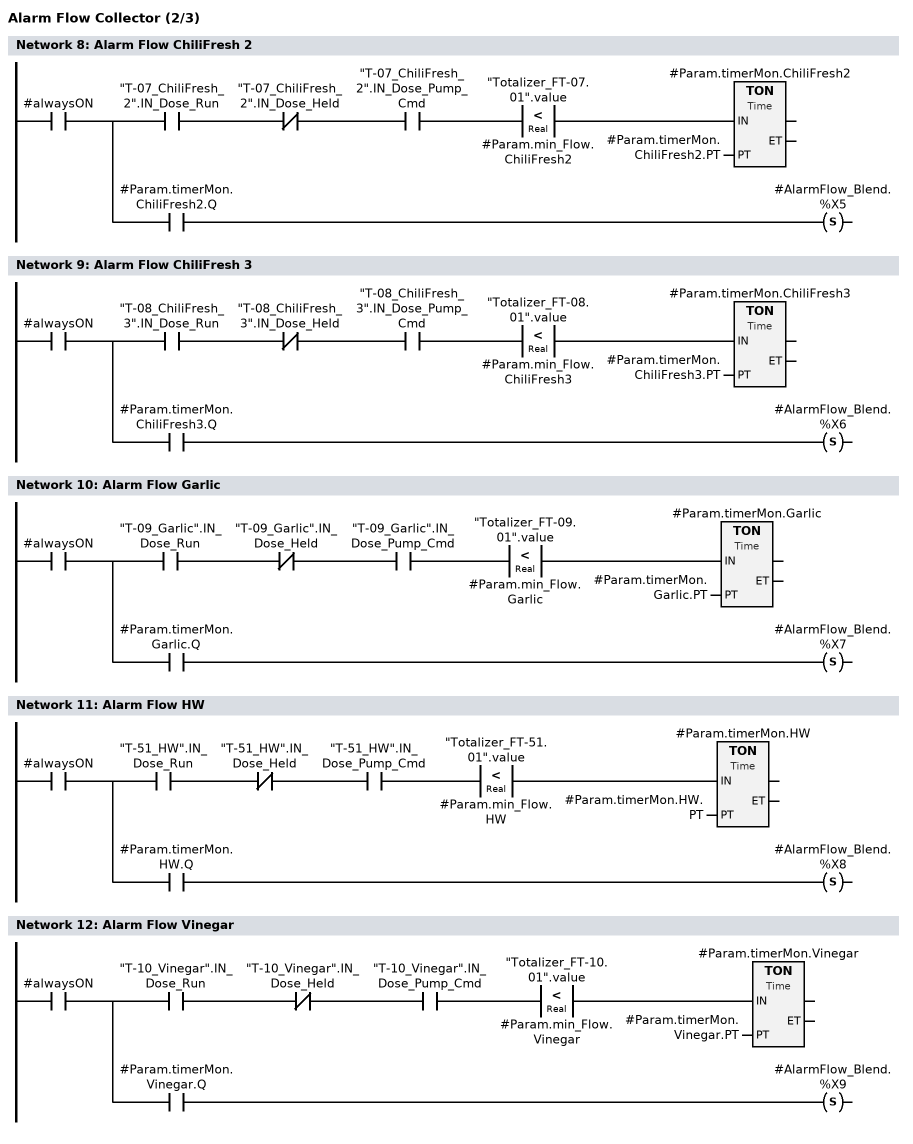
   RUNG wire#powerrail
      Contact( #alwaysON )
      wire#w1
      Contact( "T-07_ChiliFresh_2".IN_Dose_Run )
      I_Contact( "T-07_ChiliFresh_2".IN_Dose_Held )
      Contact( "T-07_ChiliFresh_2".IN_Dose_Pump_Cmd )
      { S7_Templates := "SrcType := Real" } LT_Contact(in1 := "Totalizer_FT-07.01".value, in2 := #Param.min_Flow.ChiliFresh2)
      { S7_Templates := "time_type := Time" } #Param.timerMon.ChiliFresh2.TON(pt := #Param.timerMon.ChiliFresh2.PT, et =>)
   END_RUNG
   RUNG wire#w1
      Contact( #Param.timerMon.ChiliFresh2.Q )
      S_Coil( #AlarmFlow_Blend.%X5 )
   END_RUNG
   // the same network as SCL:
   #Param.timerMon.ChiliFresh2.TON(IN := #alwaysON AND "T-07_ChiliFresh_2".IN_Dose_Run AND NOT "T-07_ChiliFresh_2".IN_Dose_Held AND "T-07_ChiliFresh_2".IN_Dose_Pump_Cmd AND ("Totalizer_FT-07.01".value < #Param.min_Flow.ChiliFresh2),
                           PT := #Param.timerMon.ChiliFresh2.PT);
   IF #alwaysON AND #Param.timerMon.ChiliFresh2.Q THEN #AlarmFlow_Blend.%X5 := TRUE; END_IF;
END_REGION

REGION Network 9: Alarm Flow ChiliFresh 3
   RUNG wire#powerrail
      Contact( #alwaysON )
      wire#w1
      Contact( "T-08_ChiliFresh_3".IN_Dose_Run )
      I_Contact( "T-08_ChiliFresh_3".IN_Dose_Held )
      Contact( "T-08_ChiliFresh_3".IN_Dose_Pump_Cmd )
      { S7_Templates := "SrcType := Real" } LT_Contact(in1 := "Totalizer_FT-08.01".value, in2 := #Param.min_Flow.ChiliFresh3)
      { S7_Templates := "time_type := Time" } #Param.timerMon.ChiliFresh3.TON(pt := #Param.timerMon.ChiliFresh3.PT, et =>)
   END_RUNG
   RUNG wire#w1
      Contact( #Param.timerMon.ChiliFresh3.Q )
      S_Coil( #AlarmFlow_Blend.%X6 )
   END_RUNG
   // the same network as SCL:
   #Param.timerMon.ChiliFresh3.TON(IN := #alwaysON AND "T-08_ChiliFresh_3".IN_Dose_Run AND NOT "T-08_ChiliFresh_3".IN_Dose_Held AND "T-08_ChiliFresh_3".IN_Dose_Pump_Cmd AND ("Totalizer_FT-08.01".value < #Param.min_Flow.ChiliFresh3),
                           PT := #Param.timerMon.ChiliFresh3.PT);
   IF #alwaysON AND #Param.timerMon.ChiliFresh3.Q THEN #AlarmFlow_Blend.%X6 := TRUE; END_IF;
END_REGION

REGION Network 10: Alarm Flow Garlic
   RUNG wire#powerrail
      Contact( #alwaysON )
      wire#w1
      Contact( "T-09_Garlic".IN_Dose_Run )
      I_Contact( "T-09_Garlic".IN_Dose_Held )
      Contact( "T-09_Garlic".IN_Dose_Pump_Cmd )
      { S7_Templates := "SrcType := Real" } LT_Contact(in1 := "Totalizer_FT-09.01".value, in2 := #Param.min_Flow.Garlic)
      { S7_Templates := "time_type := Time" } #Param.timerMon.Garlic.TON(pt := #Param.timerMon.Garlic.PT, et =>)
   END_RUNG
   RUNG wire#w1
      Contact( #Param.timerMon.Garlic.Q )
      S_Coil( #AlarmFlow_Blend.%X7 )
   END_RUNG
   // the same network as SCL:
   #Param.timerMon.Garlic.TON(IN := #alwaysON AND "T-09_Garlic".IN_Dose_Run AND NOT "T-09_Garlic".IN_Dose_Held AND "T-09_Garlic".IN_Dose_Pump_Cmd AND ("Totalizer_FT-09.01".value < #Param.min_Flow.Garlic),
                           PT := #Param.timerMon.Garlic.PT);
   IF #alwaysON AND #Param.timerMon.Garlic.Q THEN #AlarmFlow_Blend.%X7 := TRUE; END_IF;
END_REGION

REGION Network 11: Alarm Flow HW
   RUNG wire#powerrail
      Contact( #alwaysON )
      wire#w1
      Contact( "T-51_HW".IN_Dose_Run )
      I_Contact( "T-51_HW".IN_Dose_Held )
      Contact( "T-51_HW".IN_Dose_Pump_Cmd )
      { S7_Templates := "SrcType := Real" } LT_Contact(in1 := "Totalizer_FT-51.01".value, in2 := #Param.min_Flow.HW)
      { S7_Templates := "time_type := Time" } #Param.timerMon.HW.TON(pt := #Param.timerMon.HW.PT, et =>)
   END_RUNG
   RUNG wire#w1
      Contact( #Param.timerMon.HW.Q )
      S_Coil( #AlarmFlow_Blend.%X8 )
   END_RUNG
   // the same network as SCL:
   #Param.timerMon.HW.TON(IN := #alwaysON AND "T-51_HW".IN_Dose_Run AND NOT "T-51_HW".IN_Dose_Held AND "T-51_HW".IN_Dose_Pump_Cmd AND ("Totalizer_FT-51.01".value < #Param.min_Flow.HW),
                          PT := #Param.timerMon.HW.PT);
   IF #alwaysON AND #Param.timerMon.HW.Q THEN #AlarmFlow_Blend.%X8 := TRUE; END_IF;
END_REGION

REGION Network 12: Alarm Flow Vinegar
   RUNG wire#powerrail
      Contact( #alwaysON )
      wire#w1
      Contact( "T-10_Vinegar".IN_Dose_Run )
      I_Contact( "T-10_Vinegar".IN_Dose_Held )
      Contact( "T-10_Vinegar".IN_Dose_Pump_Cmd )
      { S7_Templates := "SrcType := Real" } LT_Contact(in1 := "Totalizer_FT-10.01".value, in2 := #Param.min_Flow.Vinegar)
      { S7_Templates := "time_type := Time" } #Param.timerMon.Vinegar.TON(pt := #Param.timerMon.Vinegar.PT, et =>)
   END_RUNG
   RUNG wire#w1
      Contact( #Param.timerMon.Vinegar.Q )
      S_Coil( #AlarmFlow_Blend.%X9 )
   END_RUNG
   // the same network as SCL:
   #Param.timerMon.Vinegar.TON(IN := #alwaysON AND "T-10_Vinegar".IN_Dose_Run AND NOT "T-10_Vinegar".IN_Dose_Held AND "T-10_Vinegar".IN_Dose_Pump_Cmd AND ("Totalizer_FT-10.01".value < #Param.min_Flow.Vinegar),
                           PT := #Param.timerMon.Vinegar.PT);
   IF #alwaysON AND #Param.timerMon.Vinegar.Q THEN #AlarmFlow_Blend.%X9 := TRUE; END_IF;
END_REGION

REGION Network 13: Alarm Flow Sugar
END_REGION

REGION Network 14: Alarm Flow Salt
END_REGION

REGION Network 15: Alarm Flow Prowater
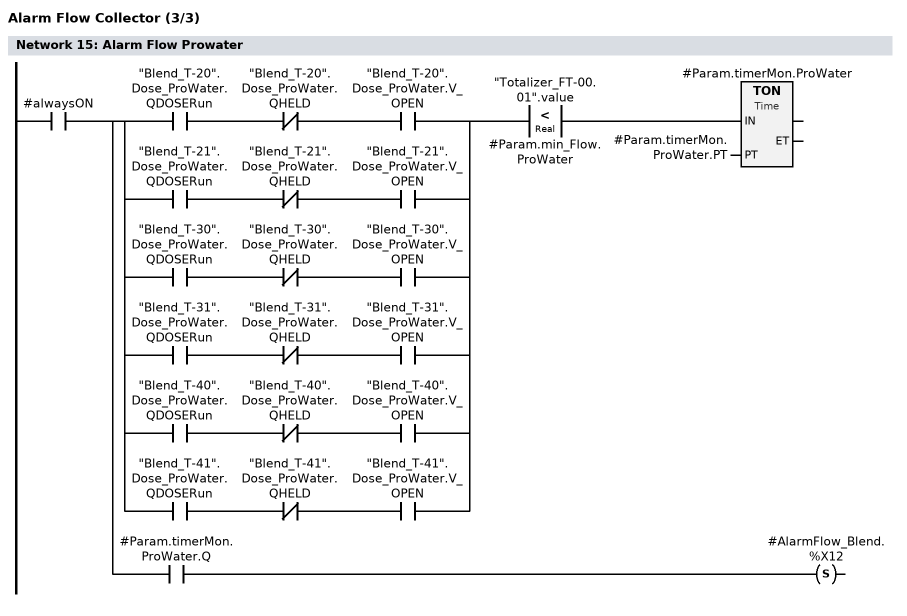
   RUNG wire#powerrail
      Contact( #alwaysON )
      wire#w1
      Contact( "Blend_T-20".Dose_ProWater.QDOSERun )
      I_Contact( "Blend_T-20".Dose_ProWater.QHELD )
      Contact( "Blend_T-20".Dose_ProWater.V_OPEN )
      wire#w2
      { S7_Templates := "SrcType := Real" } LT_Contact(in1 := "Totalizer_FT-00.01".value, in2 := #Param.min_Flow.ProWater)
      { S7_Templates := "time_type := Time" } #Param.timerMon.ProWater.TON(pt := #Param.timerMon.ProWater.PT, et =>)
   END_RUNG
   RUNG wire#w1
      Contact( "Blend_T-21".Dose_ProWater.QDOSERun )
      I_Contact( "Blend_T-21".Dose_ProWater.QHELD )
      Contact( "Blend_T-21".Dose_ProWater.V_OPEN )
   END_RUNG wire#w2
   RUNG wire#w1
      Contact( "Blend_T-30".Dose_ProWater.QDOSERun )
      I_Contact( "Blend_T-30".Dose_ProWater.QHELD )
      Contact( "Blend_T-30".Dose_ProWater.V_OPEN )
   END_RUNG wire#w2
   RUNG wire#w1
      Contact( "Blend_T-31".Dose_ProWater.QDOSERun )
      I_Contact( "Blend_T-31".Dose_ProWater.QHELD )
      Contact( "Blend_T-31".Dose_ProWater.V_OPEN )
   END_RUNG wire#w2
   RUNG wire#w1
      Contact( "Blend_T-40".Dose_ProWater.QDOSERun )
      I_Contact( "Blend_T-40".Dose_ProWater.QHELD )
      Contact( "Blend_T-40".Dose_ProWater.V_OPEN )
   END_RUNG wire#w2
   RUNG wire#w1
      Contact( "Blend_T-41".Dose_ProWater.QDOSERun )
      I_Contact( "Blend_T-41".Dose_ProWater.QHELD )
      Contact( "Blend_T-41".Dose_ProWater.V_OPEN )
   END_RUNG wire#w2
   RUNG wire#w1
      Contact( #Param.timerMon.ProWater.Q )
      S_Coil( #AlarmFlow_Blend.%X12 )
   END_RUNG
   // the same network as SCL:
   #Param.timerMon.ProWater.TON(IN := #alwaysON AND (("Blend_T-20".Dose_ProWater.QDOSERun AND NOT "Blend_T-20".Dose_ProWater.QHELD AND "Blend_T-20".Dose_ProWater.V_OPEN) OR ("Blend_T-21".Dose_ProWater.QDOSERun AND NOT "Blend_T-21".Dose_ProWater.QHELD AND "Blend_T-21".Dose_ProWater.V_OPEN) OR ("Blend_T-30".Dose_ProWater.QDOSERun AND NOT "Blend_T-30".Dose_ProWater.QHELD AND "Blend_T-30".Dose_ProWater.V_OPEN) OR ("Blend_T-31".Dose_ProWater.QDOSERun AND NOT "Blend_T-31".Dose_ProWater.QHELD AND "Blend_T-31".Dose_ProWater.V_OPEN) OR ("Blend_T-40".Dose_ProWater.QDOSERun AND NOT "Blend_T-40".Dose_ProWater.QHELD AND "Blend_T-40".Dose_ProWater.V_OPEN) OR ("Blend_T-41".Dose_ProWater.QDOSERun AND NOT "Blend_T-41".Dose_ProWater.QHELD AND "Blend_T-41".Dose_ProWater.V_OPEN)) AND ("Totalizer_FT-00.01".value < #Param.min_Flow.ProWater),
                           PT := #Param.timerMon.ProWater.PT);
   IF #alwaysON AND #Param.timerMon.ProWater.Q THEN #AlarmFlow_Blend.%X12 := TRUE; END_IF;
END_REGION
END_FUNCTION_BLOCK

FUNCTION_BLOCK "Blend_Tank"   // FB210, LAD
{ S7_Optimized_Access := 'TRUE' }
VERSION : 0.1
// stored: AutoNumber false, IsIECCheckEnabled false, IsRetainMemResEnabled false, MemoryReserve 100, SetENOAutomatically false, UDAEnableTagReadback false
   VAR_INPUT
      IN_FBAV_Header1 : Bool;
      IN_FBAV_Header2 : Bool;
      IN_FBAV_Vinegar : Bool;
      IN_FBAV_Sugar : Bool;
      IN_FBAV_Salt : Bool;
      IN_FBAV_ProWater : Bool;
      IN_FBAV_Homomixer : Bool;
      IN_FBAV_Transfer1 : Bool;
      IN_FBAV_Transfer2 : Bool;
      IN_FBAV_Transfer3 : Bool;
      IN_FBAV_Outlet : Bool;
      IN_FBAV_CIP : Bool;
      IN_FBP_Transfer1 : Bool;
      IN_FBP_Transfer1_Sp : Real;
      IN_FBP_Transfer2 : Bool;
      IN_FBP_Transfer2_Sp : Real;
      IN_FBP_Transfer3 : Bool;
      IN_FBP_Transfer3_Sp : Real;
      IN_FBP_CIP : Bool;
      IN_FBP_CIP_Sp : Real;
      IN_LT01 : Real;
      "BFT-1 Prod Req" : Bool;
      "BFT-1 Prod Line" : Bool;
      "BFT-1 CIP Enable" : Bool;
      "BFT-1 CIPLine" : Bool;
      "BFT-2 Prod Req" : Bool;
      "BFT-2 Prod Line" : Bool;
      "BFT-2 CIP Enable" : Bool;
      "BFT-2 CIPLine" : Bool;
      "BFT-3 Prod Req" : Bool;
      "BFT-3 Prod Line" : Bool;
      "BFT-3 CIP Enable" : Bool;
      "BFT-3 CIPLine" : Bool;
      "Transfer 1 Busy" : Bool;
      "Transfer 2 Busy" : Bool;
      "Transfer 3 Busy" : Bool;
      "Header 1 Available" : Bool;   // Header 1 line free
      "Header 2 Available" : Bool;   // Header 2 line free
      "Vinegar Available" : Bool;   // Vinegar line free
      "Sugar Available" : Bool;   // Sugar line free
      "Salt Available" : Bool;   // Salt line free
      "ProWater Available" : Bool;   // ProWater line free
      "Homomixer Available" : Bool;   // Homomixer line free
      IN_LDT : Date_And_Time;
      "CIP Pulse" : Bool;
      "CIP Supply ON" : Bool;
      "CIP Req OK" : Bool;
      "CIP Complete" : Bool;
      "CIP Busy" : Bool;
   END_VAR
   VAR_OUTPUT
      Out_AV_Header1 : Bool;
      Out_AV_Header2 : Bool;
      Out_AV_Vinegar : Bool;
      Out_AV_Sugar : Bool;
      Out_AV_Salt : Bool;
      Out_AV_ProWater : Bool;
      Out_AV_Homomixer : Bool;
      Out_AV_Transfer1 : Bool;
      Out_AV_Transfer2 : Bool;
      Out_AV_Transfer3 : Bool;
      Out_AV_Outlet : Bool;
      Out_AV_CIP : Bool;
      Out_P_Transfer1 : Bool;
      Out_P_Transfer1_Sp : Real;
      Out_P_Transfer2 : Bool;
      Out_P_Transfer2_Sp : Real;
      Out_P_Transfer3 : Bool;
      Out_P_Transfer3_Sp : Real;
      Out_P_CIP : Bool;
      Out_P_CIP_Sp : Real;
      Out_Agi : Bool;
      Out_Agi_Sp : Real;
      "Header 1 Req" : Bool;
      "Header 2 Req" : Bool;
      "Vinegar Req" : Bool;
      "Sugar Req" : Bool;
      "Salt Req" : Bool;
      "ProWater Req" : Bool;
      "Homomixer Req" : Bool;
      Out_CIP_Req : Bool;
      Out_CIP_Line_Open : Bool;
   END_VAR
   VAR
      Cmd : Struct
         "Ready For Transfer" : Bool;
         "CIP Tank 1" : Bool;
         "CIP Tank 2" : Bool;
         "CIP Line" : Bool;
         "Dose Head 1" : Bool;
         "Dose Head 2" : Bool;
         Agitator_Mode : Bool;   // 0: Speed Fix, 1: Speed by level
      END_STRUCT;
   END_VAR
   VAR RETAIN
      Param : Struct
         SP_Level_LL : Real := 10.0;
         SP_Level_ML : Real := 80.0;
         SP_Level_HL : Real := 100.0;
         L_Hi_Lim : Real := 100.0;
         L_Lo_Lim : Real := 0.0;
         L_Hys : Real := 2.0;
         LB_ON : Real := 20.0;
         LB_OFF : Real := 17.0;
         LB1_ON : Real := 15.0;
         LB1_OFF : Real := 10.0;
         LB2_ON : Real := 35.0;
         LB2_OFF : Real := 30.0;
         LB3_ON : Real := 65.0;
         LB3_OFF : Real := 60.0;
         SP_P1_Speed : Real := 80.0;
         SP_P2_Speed : Real := 80.0;
         SP_P3_Speed : Real := 80.0;
         SP_LB_Speed : Real := 50.0;
         SP_LB1_Speed : Real := 25.0;
         SP_LB2_Speed : Real := 50.0;
         SP_LB3_Speed : Real := 80.0;
         CIP_Tank_P_Ret_Speed : Real := 60.0;
         CIP_Ret_ON_SP : Real := 10.0;
         CIP_Ret_OFF_SP : Real := 0.0;
         Flushing_HW_Timer : Time := T#60s;
      END_STRUCT;
   END_VAR
   VAR
      State : Struct
         "Tank LL" : Bool;
         "Tank ML" : Bool;
         "Tank HL" : Bool;
         LB_ON : Bool;
         LB1_ON : Bool;
         LB2_ON : Bool;
         LB3_ON : Bool;
         "CIP Tank" : Bool;
         "CIP Tank Ena" : Bool;
         "CIP Tank Ret 1 Ena" : Bool;
         "CIP Tank Ret 2 Ena" : Bool;
         "CIP Line" : Bool;
         "CIP Line Ena" : Bool;
         "CIP Return On" : Bool;
         "Dose On Prog" : Bool;
         "Dose EN" : Bool;
         "Ready For Transfer" : Bool;
         "Ready For Transfer Ena" : Bool;
         "BFT-1 EN" : Bool;
         "BFT-2 EN" : Bool;
         "BFT-3 EN" : Bool;
         "RM Dose" : Bool;
         "Transfer 1 On Progress" : Bool;
         "Transfer 2 On Progress" : Bool;
         "Transfer 3 On Progress" : Bool;
         "DoseHead1 ON" : Bool;
         "DoseHead2 ON" : Bool;
      END_STRUCT;
      Dose : Struct
         Dose_Start : DWord;
         Dose_Pause : DWord;
         Dose_Stop : DWord;
         Dose_State : DWord;
         Dose_Tank_Available : Word;
         Dose_Prod_Ready : Word;
         Dose_Header_Req : DWord;
         Dose_EN : Word;
      END_STRUCT;
      "Dose_Level_%" : Struct
         "ChiliAwetan1%" : Real;
         "ChiliAwetan2%" : Real;
         "ChiliAwetan3%" : Real;
         "Tomato%" : Real;
         "ChiliFresh1%" : Real;
         "ChiliFresh2%" : Real;
         "ChiliFresh3%" : Real;
         "Garlic%" : Real;
         "HW%" : Real;
         "Vinegar%" : Real;
         "Sugar%" : Real;
         "Salt%" : Real;
         "ProWater%" : Real;
         "Homomixer%" : Real;
      END_STRUCT;
      Dose_Level_Lit : Struct
         ChiliAwetan1Lit : Real;
         ChiliAwetan2Lit : Real;
         ChiliAwetan3Lit : Real;
         TomatoLit : Real;
         ChiliFresh1Lit : Real;
         ChiliFresh2Lit : Real;
         ChiliFresh3Lit : Real;
         GarlicLit : Real;
         HWLit : Real;
         VinegarLit : Real;
         SugarLit : Real;
         SaltLit : Real;
         ProWaterLit : Real;
         HomomixerLit : Real;
      END_STRUCT;
      SP_Dose_Level : Struct
         ChiliAwetan1Lit : Real;
         ChiliAwetan2Lit : Real;
         ChiliAwetan3Lit : Real;
         TomatoLit : Real;
         ChiliFresh1Lit : Real;
         ChiliFresh2Lit : Real;
         ChiliFresh3Lit : Real;
         GarlicLit : Real;
         HWLit : Real;
         VinegarLit : Real;
         SugarLit : Real;
         SaltLit : Real;
         ProWaterLit : Real;
         HomomixerLit : Real;
      END_STRUCT;
      r : Struct
         PosE1 : Bool;
         PosE2 : Bool;
         PosE3 : Bool;
         PosE4 : Bool;
         PosE5 : Bool;
         PosE6 : Bool;
         PosE7 : Bool;
         PosE8 : Bool;
         PosE9 : Bool;
         PosE10 : Bool;
         PosE11 : Bool;
         PosE12 : Bool;
         PosE13 : Bool;
         PosE14 : Bool;
         PosE15 : Bool;
         PosE16 : Bool;
         PosE17 : Bool;
         PosE18 : Bool;
         PosE19 : Bool;
         PosE20 : Bool;
         PosE21 : Bool;
         PosE22 : Bool;
         PosE23 : Bool;
         PosE24 : Bool;
         PosE25 : Bool;
         PosE26 : Bool;
         PosE27 : Bool;
         PosE28 : Bool;
         PosE29 : Bool;
         PosE30 : Bool;
         PosE31 : Bool;
         PosE32 : Bool;
      END_STRUCT;
      Actuator : Struct
         P_Transfer1 : Bool;
         P_Transfer2 : Bool;
         P_Transfer3 : Bool;
         AV_Transfer1 : Bool;
         AV_Transfer2 : Bool;
         AV_Transfer3 : Bool;
         AV_Outlet : Bool;
         AV_CIP_Tank : Bool;
      END_STRUCT;
      SP_ChiliAwetan1 : "RawDose";
      SP_ChiliAwetan2 : "RawDose";
      SP_ChiliAwetan3 : "RawDose";
      SP_Tomato : "RawDose";
      SP_ChiliFresh1 : "RawDose";
      SP_ChiliFresh2 : "RawDose";
      SP_ChiliFresh3 : "RawDose";
      SP_Garlic : "RawDose";
      SP_HW : "Raw_Pulse";
      SP_Vinegar : "RawDose";
      SP_Sugar : "RawDose";
      SP_Salt : "RawDose";
      SP_ProWater : "Raw_Pulse";
      SP_Homomixer : "RawDose";
      Dose_ChiliAwetan1 { S7_SetPoint := 'True'} : "DOSE";
      Dose_ChiliAwetan2 { S7_SetPoint := 'True'} : "DOSE";
      Dose_ChiliAwetan3 { S7_SetPoint := 'True'} : "DOSE";
      Dose_Tomato { S7_SetPoint := 'True'} : "DOSE";
      Dose_ChiliFresh1 { S7_SetPoint := 'True'} : "DOSE";
      Dose_ChiliFresh2 { S7_SetPoint := 'True'} : "DOSE";
      Dose_ChiliFresh3 { S7_SetPoint := 'True'} : "DOSE";
      Dose_Garlic { S7_SetPoint := 'True'} : "DOSE";
      Dose_HW { S7_SetPoint := 'True'} : "DOSE";
      Dose_Vinegar { S7_SetPoint := 'True'} : "DOSE";
      Dose_Sugar { S7_SetPoint := 'True'} : "DOSE";
      Dose_Salt { S7_SetPoint := 'True'} : "DOSE";
      Dose_ProWater { S7_SetPoint := 'True'} : "DOSE";
      Dose_Homomixer { S7_SetPoint := 'True'} : "DOSE";
      AlwaysON { S7_SetPoint := 'True'} : Bool;
      L_Hys_Abs { S7_SetPoint := 'True'} : Real;
      Hys_Level_HL : Real;
      Hys_Level_ML : Real;
      Hys_Level_LL : Real;
      TimerOff_Valve_Out : TON_TIME;
      TimerOff_Valve_P_1 { S7_SetPoint := 'True'} : TON_TIME;
      TimerOff_Valve_P_2 { S7_SetPoint := 'True'} : TON_TIME;
      TimerOff_Valve_P_3 { S7_SetPoint := 'True'} : TON_TIME;
      TimerOff_Valve_P_CIP { S7_SetPoint := 'True'} : TON_TIME;
   END_VAR
   VAR RETAIN
      Last_Dose_Qty : Struct
         ChiliAwetan1 : Real;
         ChiliAwetan2 : Real;
         ChiliAwetan3 : Real;
         Tomato : Real;
         ChiliFresh1 : Real;
         ChiliFresh2 : Real;
         ChiliFresh3 : Real;
         Garlic : Real;
         HW : Real;
         Vinegar : Real;
         Sugar : Real;
         Salt : Real;
         ProWater : Real;
         Homomixer : Real;
      END_STRUCT;
   END_VAR
   VAR
      "HW Flushing" : Struct
         Status : Struct
            "Flush to Blend" : Bool;
            "Flush to Drain" : Bool;
            Drain : Bool;
            Done : Bool;
         END_STRUCT;
         Qty : Struct
            "Flush to Blend Qty" : Real;
            "Flush to Drain Qty" : Real;
            "Flush to Blend Act" : Real;
            "Flush to Drain Act" : Real;
         END_STRUCT;
         TimeDrain_SP : DInt;
         Cmd_Start_Drain : Bool;
         Cmd_Stop_Drain : Bool;
         DrainTime : TONR_TIME;
      END_STRUCT;
      PumpTF1_OnDelay : TON_TIME;
      PumpTF2_OnDelay { S7_SetPoint := 'True'} : TON_TIME;
      PumpTF3_OnDelay { S7_SetPoint := 'True'} : TON_TIME;
   END_VAR
   VAR RETAIN
      TimerON : Struct
         TimerON_1 : TON_TIME;
         TimerON_2 { S7_SetPoint := 'True'} : TON_TIME;
         TimerON_3 { S7_SetPoint := 'True'} : TON_TIME;
         TimerON_4 { S7_SetPoint := 'True'} : TON_TIME;
         TimerON_5 { S7_SetPoint := 'True'} : TON_TIME;
         TimerON_6 { S7_SetPoint := 'True'} : TON_TIME;
         TimerON_7 { S7_SetPoint := 'True'} : TON_TIME;
         TimerON_8 { S7_SetPoint := 'True'} : TON_TIME;
      END_STRUCT;
      TimerOFF : Struct
         TimerOFF_1 : TOF_TIME;
         TimerOFF_2 { S7_SetPoint := 'True'} : TOF_TIME;
         TimerOFF_3 { S7_SetPoint := 'True'} : TOF_TIME;
         TimerOFF_4 { S7_SetPoint := 'True'} : TOF_TIME;
         TimerOFF_5 { S7_SetPoint := 'True'} : TOF_TIME;
         TimerOFF_6 { S7_SetPoint := 'True'} : TOF_TIME;
         TimerOFF_7 { S7_SetPoint := 'True'} : TOF_TIME;
         TimerOFF_8 { S7_SetPoint := 'True'} : TOF_TIME;
      END_STRUCT;
   END_VAR
   // SP_ProWater.Para."SP_Qty_Fine%" := 10.0;
   // SP_Homomixer.Dose_SP := 10.0;
   // TimerON.TimerON_1.PT := T#8s;
   // TimerON.TimerON_2.PT := T#8s;
   // TimerON.TimerON_3.PT := T#10s;
   // TimerON.TimerON_4.PT := T#10s;
   // TimerON.TimerON_5.PT := T#10s;
   // TimerON.TimerON_6.PT := T#10s;
   // TimerON.TimerON_7.PT := T#10s;
   // TimerON.TimerON_8.PT := T#10s;
   // TimerOFF.TimerOFF_1.PT := T#10s;
   // TimerOFF.TimerOFF_2.PT := T#10s;
   // TimerOFF.TimerOFF_3.PT := T#10s;
   // TimerOFF.TimerOFF_4.PT := T#10s;
   // TimerOFF.TimerOFF_5.PT := T#10s;
   // TimerOFF.TimerOFF_6.PT := T#10s;
   // TimerOFF.TimerOFF_7.PT := T#10s;
   // TimerOFF.TimerOFF_8.PT := T#10s;
   VAR_TEMP   // added for the SCL form of the ladder/FBD networks
      _w1 : Bool;
      _w2 : Bool;
      _w3 : Bool;
      _w4 : Bool;
      _w5 : Bool;
      _w6 : Bool;
   END_VAR
BEGIN

REGION Network 2: Always ON
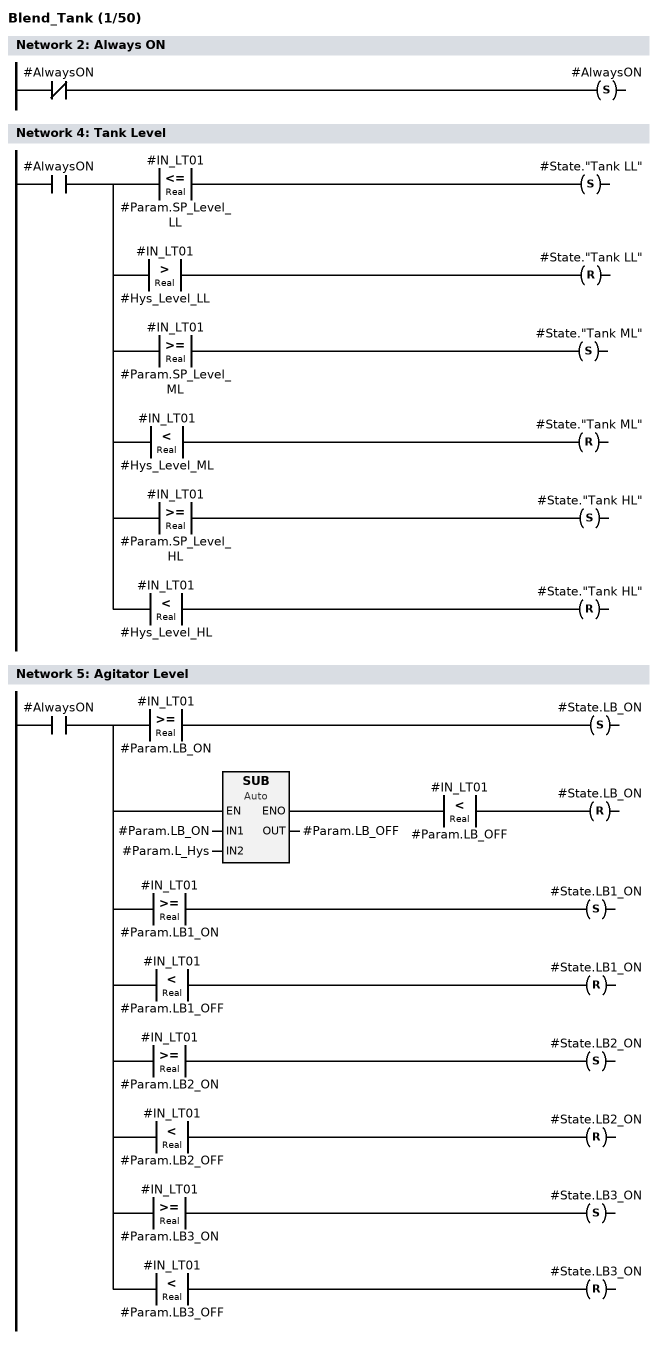
   RUNG wire#powerrail
      I_Contact( #AlwaysON )
      S_Coil( #AlwaysON )
   END_RUNG
   // the same network as SCL:
   IF NOT #AlwaysON THEN #AlwaysON := TRUE; END_IF;
END_REGION

NETWORK
TITLE = Hys Calculation
//Level Hys Absolute
      L     #Param.L_Hi_Lim;
      L     #Param.L_Lo_Lim;
      -R;
      L     100.0;
      /R;
      L     #Param.L_Hys;
      *R;
      T     #L_Hys_Abs;
//Tank High Level
      L     #Param.SP_Level_HL;
      L     #L_Hys_Abs;
      -R;
      T     #Hys_Level_HL;
//Tank Mid Level
      L     #Param.SP_Level_ML;
      L     #L_Hys_Abs;
      -R;
      T     #Hys_Level_ML;
//Tank Low Level
      L     #Param.SP_Level_LL;
      L     #L_Hys_Abs;
      +R;
      T     #Hys_Level_LL;


REGION Network 4: Tank Level
   RUNG wire#powerrail
      Contact( #AlwaysON )
      wire#w1
      { S7_Templates := "SrcType := Real" } LE_Contact(in1 := #IN_LT01, in2 := #Param.SP_Level_LL)
      S_Coil( #State."Tank LL" )
   END_RUNG
   RUNG wire#w1
      { S7_Templates := "SrcType := Real" } GT_Contact(in1 := #IN_LT01, in2 := #Hys_Level_LL)
      R_Coil( #State."Tank LL" )
   END_RUNG
   RUNG wire#w1
      { S7_Templates := "SrcType := Real" } GE_Contact(in1 := #IN_LT01, in2 := #Param.SP_Level_ML)
      S_Coil( #State."Tank ML" )
   END_RUNG
   RUNG wire#w1
      { S7_Templates := "SrcType := Real" } LT_Contact(in1 := #IN_LT01, in2 := #Hys_Level_ML)
      R_Coil( #State."Tank ML" )
   END_RUNG
   RUNG wire#w1
      { S7_Templates := "SrcType := Real" } GE_Contact(in1 := #IN_LT01, in2 := #Param.SP_Level_HL)
      S_Coil( #State."Tank HL" )
   END_RUNG
   RUNG wire#w1
      { S7_Templates := "SrcType := Real" } LT_Contact(in1 := #IN_LT01, in2 := #Hys_Level_HL)
      R_Coil( #State."Tank HL" )
   END_RUNG
   // the same network as SCL:
   IF #AlwaysON AND (#IN_LT01 <= #Param.SP_Level_LL) THEN #State."Tank LL" := TRUE; END_IF;
   IF #AlwaysON AND (#IN_LT01 > #Hys_Level_LL) THEN #State."Tank LL" := FALSE; END_IF;
   IF #AlwaysON AND (#IN_LT01 >= #Param.SP_Level_ML) THEN #State."Tank ML" := TRUE; END_IF;
   IF #AlwaysON AND (#IN_LT01 < #Hys_Level_ML) THEN #State."Tank ML" := FALSE; END_IF;
   IF #AlwaysON AND (#IN_LT01 >= #Param.SP_Level_HL) THEN #State."Tank HL" := TRUE; END_IF;
   IF #AlwaysON AND (#IN_LT01 < #Hys_Level_HL) THEN #State."Tank HL" := FALSE; END_IF;
END_REGION

REGION Network 5: Agitator Level
   RUNG wire#powerrail
      Contact( #AlwaysON )
      wire#w1
      { S7_Templates := "SrcType := Real" } GE_Contact(in1 := #IN_LT01, in2 := #Param.LB_ON)
      S_Coil( #State.LB_ON )
   END_RUNG
   RUNG wire#w1
      Sub(in1 := #Param.LB_ON, in2 := #Param.L_Hys, out => #Param.LB_OFF)
      { S7_Templates := "SrcType := Real" } LT_Contact(in1 := #IN_LT01, in2 := #Param.LB_OFF)
      R_Coil( #State.LB_ON )
   END_RUNG
   RUNG wire#w1
      { S7_Templates := "SrcType := Real" } GE_Contact(in1 := #IN_LT01, in2 := #Param.LB1_ON)
      S_Coil( #State.LB1_ON )
   END_RUNG
   RUNG wire#w1
      { S7_Templates := "SrcType := Real" } LT_Contact(in1 := #IN_LT01, in2 := #Param.LB1_OFF)
      R_Coil( #State.LB1_ON )
   END_RUNG
   RUNG wire#w1
      { S7_Templates := "SrcType := Real" } GE_Contact(in1 := #IN_LT01, in2 := #Param.LB2_ON)
      S_Coil( #State.LB2_ON )
   END_RUNG
   RUNG wire#w1
      { S7_Templates := "SrcType := Real" } LT_Contact(in1 := #IN_LT01, in2 := #Param.LB2_OFF)
      R_Coil( #State.LB2_ON )
   END_RUNG
   RUNG wire#w1
      { S7_Templates := "SrcType := Real" } GE_Contact(in1 := #IN_LT01, in2 := #Param.LB3_ON)
      S_Coil( #State.LB3_ON )
   END_RUNG
   RUNG wire#w1
      { S7_Templates := "SrcType := Real" } LT_Contact(in1 := #IN_LT01, in2 := #Param.LB3_OFF)
      R_Coil( #State.LB3_ON )
   END_RUNG
   // the same network as SCL:
   IF #AlwaysON AND (#IN_LT01 >= #Param.LB_ON) THEN #State.LB_ON := TRUE; END_IF;
   IF #AlwaysON THEN #Param.LB_OFF := #Param.LB_ON - #Param.L_Hys; END_IF;
   IF #AlwaysON AND (#IN_LT01 < #Param.LB_OFF) THEN #State.LB_ON := FALSE; END_IF;
   IF #AlwaysON AND (#IN_LT01 >= #Param.LB1_ON) THEN #State.LB1_ON := TRUE; END_IF;
   IF #AlwaysON AND (#IN_LT01 < #Param.LB1_OFF) THEN #State.LB1_ON := FALSE; END_IF;
   IF #AlwaysON AND (#IN_LT01 >= #Param.LB2_ON) THEN #State.LB2_ON := TRUE; END_IF;
   IF #AlwaysON AND (#IN_LT01 < #Param.LB2_OFF) THEN #State.LB2_ON := FALSE; END_IF;
   IF #AlwaysON AND (#IN_LT01 >= #Param.LB3_ON) THEN #State.LB3_ON := TRUE; END_IF;
   IF #AlwaysON AND (#IN_LT01 < #Param.LB3_OFF) THEN #State.LB3_ON := FALSE; END_IF;
END_REGION

REGION Network 6: Agitator ON-OFF
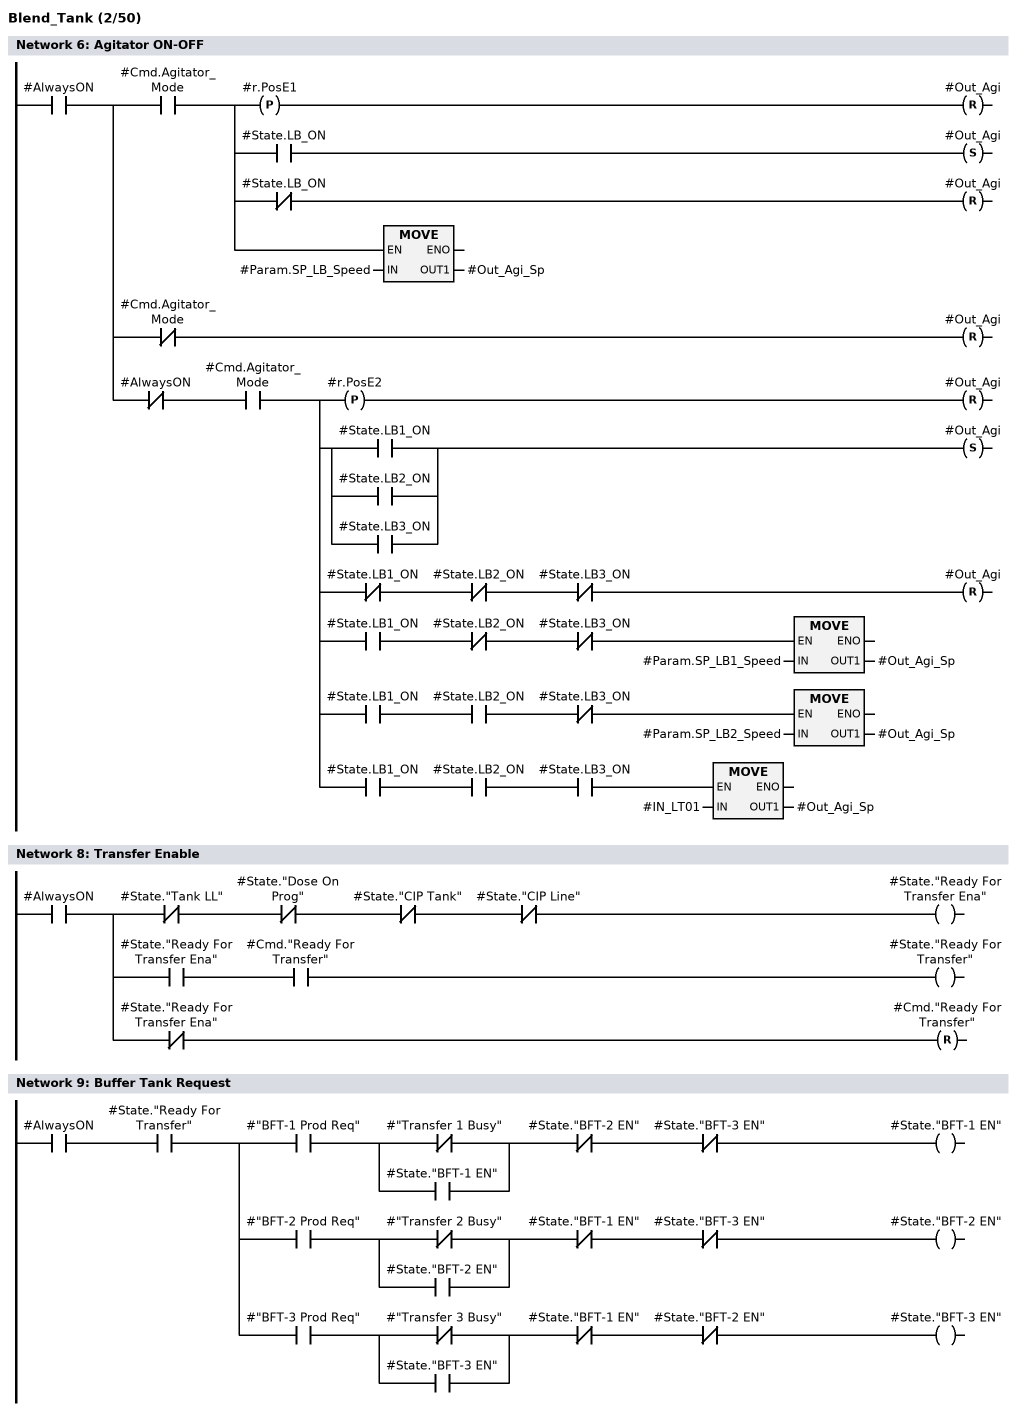
   RUNG wire#powerrail
      Contact( #AlwaysON )
      wire#w1
      Contact( #Cmd.Agitator_Mode )
      wire#w2
      P_Trig( #r.PosE1 )
      R_Coil( #Out_Agi )
   END_RUNG
   RUNG wire#w2
      Contact( #State.LB_ON )
      S_Coil( #Out_Agi )
   END_RUNG
   RUNG wire#w2
      I_Contact( #State.LB_ON )
      R_Coil( #Out_Agi )
   END_RUNG
   RUNG wire#w2
      Move(in := #Param.SP_LB_Speed, out1 => #Out_Agi_Sp)
   END_RUNG
   RUNG wire#w1
      I_Contact( #Cmd.Agitator_Mode )
      R_Coil( #Out_Agi )
   END_RUNG
   RUNG wire#w1
      I_Contact( #AlwaysON )
      Contact( #Cmd.Agitator_Mode )
      wire#w3
      P_Trig( #r.PosE2 )
      R_Coil( #Out_Agi )
   END_RUNG
   RUNG wire#w3
      Contact( #State.LB1_ON )
      wire#w4
      S_Coil( #Out_Agi )
   END_RUNG
   RUNG wire#w3
      Contact( #State.LB2_ON )
   END_RUNG wire#w4
   RUNG wire#w3
      Contact( #State.LB3_ON )
   END_RUNG wire#w4
   RUNG wire#w3
      I_Contact( #State.LB1_ON )
      I_Contact( #State.LB2_ON )
      I_Contact( #State.LB3_ON )
      R_Coil( #Out_Agi )
   END_RUNG
   RUNG wire#w3
      Contact( #State.LB1_ON )
      I_Contact( #State.LB2_ON )
      I_Contact( #State.LB3_ON )
      Move(in := #Param.SP_LB1_Speed, out1 => #Out_Agi_Sp)
   END_RUNG
   RUNG wire#w3
      Contact( #State.LB1_ON )
      Contact( #State.LB2_ON )
      I_Contact( #State.LB3_ON )
      Move(in := #Param.SP_LB2_Speed, out1 => #Out_Agi_Sp)
   END_RUNG
   RUNG wire#w3
      Contact( #State.LB1_ON )
      Contact( #State.LB2_ON )
      Contact( #State.LB3_ON )
      Move(in := #IN_LT01, out1 => #Out_Agi_Sp)
   END_RUNG
   // the same network as SCL:
   #_w1 := #AlwaysON AND #Cmd.Agitator_Mode;
   #_w2 := #_w1 AND NOT #r.PosE1;   // rising edge
   #r.PosE1 := #_w1;
   IF #_w2 THEN #Out_Agi := FALSE; END_IF;
   IF #_w1 AND #State.LB_ON THEN #Out_Agi := TRUE; END_IF;
   IF #_w1 AND NOT #State.LB_ON THEN #Out_Agi := FALSE; END_IF;
   IF #_w1 THEN #Out_Agi_Sp := #Param.SP_LB_Speed; END_IF;
   IF #AlwaysON AND NOT #Cmd.Agitator_Mode THEN #Out_Agi := FALSE; END_IF;
   #_w3 := #AlwaysON AND NOT #AlwaysON AND #Cmd.Agitator_Mode;
   #_w4 := #_w3 AND NOT #r.PosE2;   // rising edge
   #r.PosE2 := #_w3;
   IF #_w4 THEN #Out_Agi := FALSE; END_IF;
   IF #_w3 AND (#State.LB1_ON OR #State.LB2_ON OR #State.LB3_ON) THEN #Out_Agi := TRUE; END_IF;
   IF #_w3 AND NOT #State.LB1_ON AND NOT #State.LB2_ON AND NOT #State.LB3_ON THEN #Out_Agi := FALSE; END_IF;
   IF #_w3 AND #State.LB1_ON AND NOT #State.LB2_ON AND NOT #State.LB3_ON THEN
       #Out_Agi_Sp := #Param.SP_LB1_Speed;
   END_IF;
   IF #_w3 AND #State.LB1_ON AND #State.LB2_ON AND NOT #State.LB3_ON THEN
       #Out_Agi_Sp := #Param.SP_LB2_Speed;
   END_IF;
   IF #_w3 AND #State.LB1_ON AND #State.LB2_ON AND #State.LB3_ON THEN #Out_Agi_Sp := #IN_LT01; END_IF;
END_REGION

REGION Network 8: Transfer Enable
   RUNG wire#powerrail
      Contact( #AlwaysON )
      wire#w1
      I_Contact( #State."Tank LL" )
      I_Contact( #State."Dose On Prog" )
      I_Contact( #State."CIP Tank" )
      I_Contact( #State."CIP Line" )
      Coil( #State."Ready For Transfer Ena" )
   END_RUNG
   RUNG wire#w1
      Contact( #State."Ready For Transfer Ena" )
      Contact( #Cmd."Ready For Transfer" )
      Coil( #State."Ready For Transfer" )
   END_RUNG
   RUNG wire#w1
      I_Contact( #State."Ready For Transfer Ena" )
      R_Coil( #Cmd."Ready For Transfer" )
   END_RUNG
   // the same network as SCL:
   #State."Ready For Transfer Ena" := #AlwaysON AND NOT #State."Tank LL" AND NOT #State."Dose On Prog" AND NOT #State."CIP Tank" AND NOT #State."CIP Line";
   #State."Ready For Transfer" := #AlwaysON AND #State."Ready For Transfer Ena" AND #Cmd."Ready For Transfer";
   IF #AlwaysON AND NOT #State."Ready For Transfer Ena" THEN #Cmd."Ready For Transfer" := FALSE; END_IF;
END_REGION

REGION Network 9: Buffer Tank Request
   RUNG wire#powerrail
      Contact( #AlwaysON )
      Contact( #State."Ready For Transfer" )
      wire#w1
      Contact( #"BFT-1 Prod Req" )
      wire#w2
      I_Contact( #"Transfer 1 Busy" )
      wire#w3
      I_Contact( #State."BFT-2 EN" )
      I_Contact( #State."BFT-3 EN" )
      Coil( #State."BFT-1 EN" )
   END_RUNG
   RUNG wire#w2
      Contact( #State."BFT-1 EN" )
   END_RUNG wire#w3
   RUNG wire#w1
      Contact( #"BFT-2 Prod Req" )
      wire#w4
      I_Contact( #"Transfer 2 Busy" )
      wire#w5
      I_Contact( #State."BFT-1 EN" )
      I_Contact( #State."BFT-3 EN" )
      Coil( #State."BFT-2 EN" )
   END_RUNG
   RUNG wire#w4
      Contact( #State."BFT-2 EN" )
   END_RUNG wire#w5
   RUNG wire#w1
      Contact( #"BFT-3 Prod Req" )
      wire#w6
      I_Contact( #"Transfer 3 Busy" )
      wire#w7
      I_Contact( #State."BFT-1 EN" )
      I_Contact( #State."BFT-2 EN" )
      Coil( #State."BFT-3 EN" )
   END_RUNG
   RUNG wire#w6
      Contact( #State."BFT-3 EN" )
   END_RUNG wire#w7
   // the same network as SCL:
   #_w1 := #AlwaysON AND #State."Ready For Transfer";
   #State."BFT-1 EN" := #_w1 AND #"BFT-1 Prod Req" AND (NOT #"Transfer 1 Busy" OR #State."BFT-1 EN") AND NOT #State."BFT-2 EN" AND NOT #State."BFT-3 EN";
   #State."BFT-2 EN" := #_w1 AND #"BFT-2 Prod Req" AND (NOT #"Transfer 2 Busy" OR #State."BFT-2 EN") AND NOT #State."BFT-1 EN" AND NOT #State."BFT-3 EN";
   #State."BFT-3 EN" := #_w1 AND #"BFT-3 Prod Req" AND (NOT #"Transfer 3 Busy" OR #State."BFT-3 EN") AND NOT #State."BFT-1 EN" AND NOT #State."BFT-2 EN";
END_REGION

REGION Network 10: Buffer Tank Transfer Progress
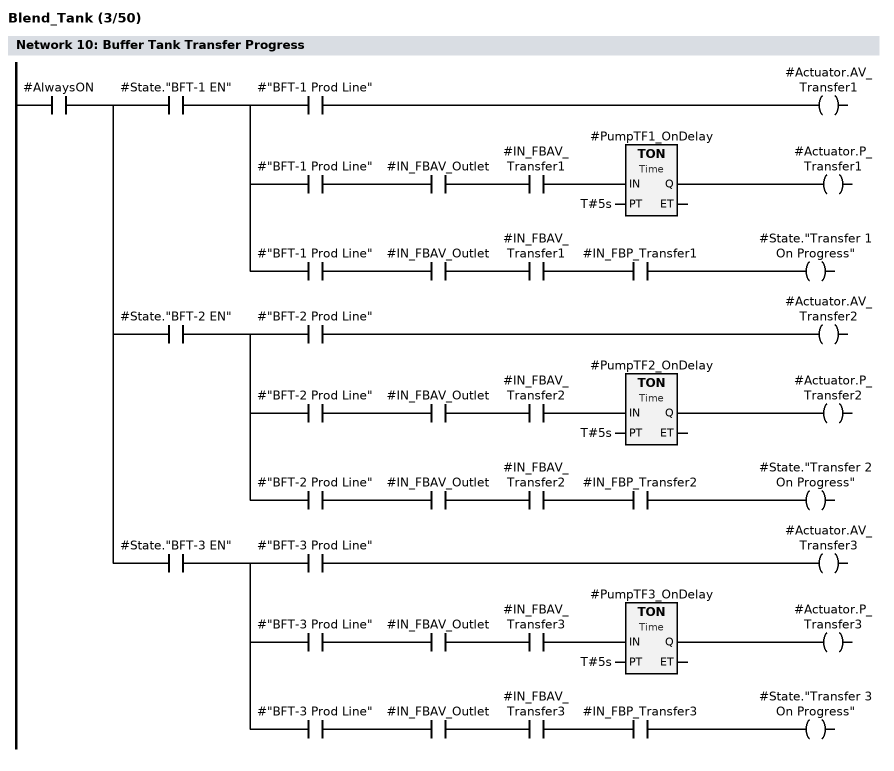
   RUNG wire#powerrail
      Contact( #AlwaysON )
      wire#w1
      Contact( #State."BFT-1 EN" )
      wire#w2
      Contact( #"BFT-1 Prod Line" )
      Coil( #Actuator.AV_Transfer1 )
   END_RUNG
   RUNG wire#w2
      Contact( #"BFT-1 Prod Line" )
      Contact( #IN_FBAV_Outlet )
      Contact( #IN_FBAV_Transfer1 )
      { S7_Templates := "time_type := Time" } #PumpTF1_OnDelay.TON(pt := T#5s, et =>)
      Coil( #Actuator.P_Transfer1 )
   END_RUNG
   RUNG wire#w2
      Contact( #"BFT-1 Prod Line" )
      Contact( #IN_FBAV_Outlet )
      Contact( #IN_FBAV_Transfer1 )
      Contact( #IN_FBP_Transfer1 )
      Coil( #State."Transfer 1 On Progress" )
   END_RUNG
   RUNG wire#w1
      Contact( #State."BFT-2 EN" )
      wire#w3
      Contact( #"BFT-2 Prod Line" )
      Coil( #Actuator.AV_Transfer2 )
   END_RUNG
   RUNG wire#w3
      Contact( #"BFT-2 Prod Line" )
      Contact( #IN_FBAV_Outlet )
      Contact( #IN_FBAV_Transfer2 )
      { S7_Templates := "time_type := Time" } #PumpTF2_OnDelay.TON(pt := T#5s, et =>)
      Coil( #Actuator.P_Transfer2 )
   END_RUNG
   RUNG wire#w3
      Contact( #"BFT-2 Prod Line" )
      Contact( #IN_FBAV_Outlet )
      Contact( #IN_FBAV_Transfer2 )
      Contact( #IN_FBP_Transfer2 )
      Coil( #State."Transfer 2 On Progress" )
   END_RUNG
   RUNG wire#w1
      Contact( #State."BFT-3 EN" )
      wire#w4
      Contact( #"BFT-3 Prod Line" )
      Coil( #Actuator.AV_Transfer3 )
   END_RUNG
   RUNG wire#w4
      Contact( #"BFT-3 Prod Line" )
      Contact( #IN_FBAV_Outlet )
      Contact( #IN_FBAV_Transfer3 )
      { S7_Templates := "time_type := Time" } #PumpTF3_OnDelay.TON(pt := T#5s, et =>)
      Coil( #Actuator.P_Transfer3 )
   END_RUNG
   RUNG wire#w4
      Contact( #"BFT-3 Prod Line" )
      Contact( #IN_FBAV_Outlet )
      Contact( #IN_FBAV_Transfer3 )
      Contact( #IN_FBP_Transfer3 )
      Coil( #State."Transfer 3 On Progress" )
   END_RUNG
   // the same network as SCL:
   #_w1 := #AlwaysON AND #State."BFT-1 EN";
   #Actuator.AV_Transfer1 := #_w1 AND #"BFT-1 Prod Line";
   #PumpTF1_OnDelay(IN := #_w1 AND #"BFT-1 Prod Line" AND #IN_FBAV_Outlet AND #IN_FBAV_Transfer1, PT := T#5s);   // TON
   #Actuator.P_Transfer1 := #PumpTF1_OnDelay.Q;
   #State."Transfer 1 On Progress" := #_w1 AND #"BFT-1 Prod Line" AND #IN_FBAV_Outlet AND #IN_FBAV_Transfer1 AND #IN_FBP_Transfer1;
   #_w2 := #AlwaysON AND #State."BFT-2 EN";
   #Actuator.AV_Transfer2 := #_w2 AND #"BFT-2 Prod Line";
   #PumpTF2_OnDelay(IN := #_w2 AND #"BFT-2 Prod Line" AND #IN_FBAV_Outlet AND #IN_FBAV_Transfer2, PT := T#5s);   // TON
   #Actuator.P_Transfer2 := #PumpTF2_OnDelay.Q;
   #State."Transfer 2 On Progress" := #_w2 AND #"BFT-2 Prod Line" AND #IN_FBAV_Outlet AND #IN_FBAV_Transfer2 AND #IN_FBP_Transfer2;
   #_w3 := #AlwaysON AND #State."BFT-3 EN";
   #Actuator.AV_Transfer3 := #_w3 AND #"BFT-3 Prod Line";
   #PumpTF3_OnDelay(IN := #_w3 AND #"BFT-3 Prod Line" AND #IN_FBAV_Outlet AND #IN_FBAV_Transfer3, PT := T#5s);   // TON
   #Actuator.P_Transfer3 := #PumpTF3_OnDelay.Q;
   #State."Transfer 3 On Progress" := #_w3 AND #"BFT-3 Prod Line" AND #IN_FBAV_Outlet AND #IN_FBAV_Transfer3 AND #IN_FBP_Transfer3;
END_REGION

REGION Network 12: Command CIP
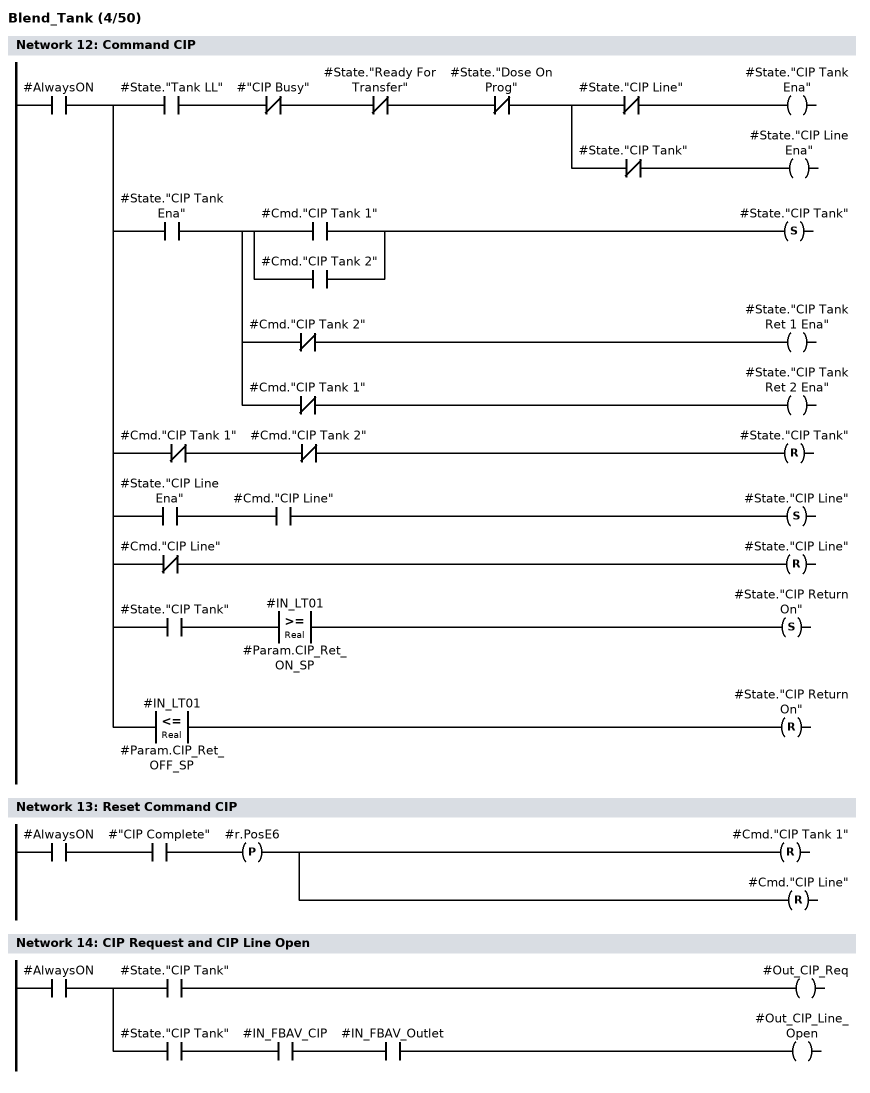
   RUNG wire#powerrail
      Contact( #AlwaysON )
      wire#w1
      Contact( #State."Tank LL" )
      I_Contact( #"CIP Busy" )
      I_Contact( #State."Ready For Transfer" )
      I_Contact( #State."Dose On Prog" )
      wire#w2
      I_Contact( #State."CIP Line" )
      Coil( #State."CIP Tank Ena" )
   END_RUNG
   RUNG wire#w2
      I_Contact( #State."CIP Tank" )
      Coil( #State."CIP Line Ena" )
   END_RUNG
   RUNG wire#w1
      Contact( #State."CIP Tank Ena" )
      wire#w3
      Contact( #Cmd."CIP Tank 1" )
      wire#w4
      S_Coil( #State."CIP Tank" )
   END_RUNG
   RUNG wire#w3
      Contact( #Cmd."CIP Tank 2" )
   END_RUNG wire#w4
   RUNG wire#w3
      I_Contact( #Cmd."CIP Tank 2" )
      Coil( #State."CIP Tank Ret 1 Ena" )
   END_RUNG
   RUNG wire#w3
      I_Contact( #Cmd."CIP Tank 1" )
      Coil( #State."CIP Tank Ret 2 Ena" )
   END_RUNG
   RUNG wire#w1
      I_Contact( #Cmd."CIP Tank 1" )
      I_Contact( #Cmd."CIP Tank 2" )
      R_Coil( #State."CIP Tank" )
   END_RUNG
   RUNG wire#w1
      Contact( #State."CIP Line Ena" )
      Contact( #Cmd."CIP Line" )
      S_Coil( #State."CIP Line" )
   END_RUNG
   RUNG wire#w1
      I_Contact( #Cmd."CIP Line" )
      R_Coil( #State."CIP Line" )
   END_RUNG
   RUNG wire#w1
      Contact( #State."CIP Tank" )
      { S7_Templates := "SrcType := Real" } GE_Contact(in1 := #IN_LT01, in2 := #Param.CIP_Ret_ON_SP)
      S_Coil( #State."CIP Return On" )
   END_RUNG
   RUNG wire#w1
      { S7_Templates := "SrcType := Real" } LE_Contact(in1 := #IN_LT01, in2 := #Param.CIP_Ret_OFF_SP)
      R_Coil( #State."CIP Return On" )
   END_RUNG
   // the same network as SCL:
   #_w1 := #AlwaysON AND #State."Tank LL" AND NOT #"CIP Busy" AND NOT #State."Ready For Transfer" AND NOT #State."Dose On Prog";
   #State."CIP Tank Ena" := #_w1 AND NOT #State."CIP Line";
   #State."CIP Line Ena" := #_w1 AND NOT #State."CIP Tank";
   #_w2 := #AlwaysON AND #State."CIP Tank Ena";
   IF #_w2 AND (#Cmd."CIP Tank 1" OR #Cmd."CIP Tank 2") THEN #State."CIP Tank" := TRUE; END_IF;
   #State."CIP Tank Ret 1 Ena" := #_w2 AND NOT #Cmd."CIP Tank 2";
   #State."CIP Tank Ret 2 Ena" := #_w2 AND NOT #Cmd."CIP Tank 1";
   IF #AlwaysON AND NOT #Cmd."CIP Tank 1" AND NOT #Cmd."CIP Tank 2" THEN #State."CIP Tank" := FALSE; END_IF;
   IF #AlwaysON AND #State."CIP Line Ena" AND #Cmd."CIP Line" THEN #State."CIP Line" := TRUE; END_IF;
   IF #AlwaysON AND NOT #Cmd."CIP Line" THEN #State."CIP Line" := FALSE; END_IF;
   IF #AlwaysON AND #State."CIP Tank" AND (#IN_LT01 >= #Param.CIP_Ret_ON_SP) THEN
       #State."CIP Return On" := TRUE;
   END_IF;
   IF #AlwaysON AND (#IN_LT01 <= #Param.CIP_Ret_OFF_SP) THEN #State."CIP Return On" := FALSE; END_IF;
END_REGION

REGION Network 13: Reset Command CIP
   RUNG wire#powerrail
      Contact( #AlwaysON )
      Contact( #"CIP Complete" )
      P_Trig( #r.PosE6 )
      wire#w1
      R_Coil( #Cmd."CIP Tank 1" )
   END_RUNG
   RUNG wire#w1
      R_Coil( #Cmd."CIP Line" )
   END_RUNG
   // the same network as SCL:
   #_w1 := #AlwaysON AND #"CIP Complete";
   #_w2 := #_w1 AND NOT #r.PosE6;   // rising edge
   #r.PosE6 := #_w1;
   IF #_w2 THEN
       #Cmd."CIP Tank 1" := FALSE;
       #Cmd."CIP Line" := FALSE;
   END_IF;
END_REGION

REGION Network 14: CIP Request and CIP Line Open
   RUNG wire#powerrail
      Contact( #AlwaysON )
      wire#w1
      Contact( #State."CIP Tank" )
      Coil( #Out_CIP_Req )
   END_RUNG
   RUNG wire#w1
      Contact( #State."CIP Tank" )
      Contact( #IN_FBAV_CIP )
      Contact( #IN_FBAV_Outlet )
      Coil( #Out_CIP_Line_Open )
   END_RUNG
   // the same network as SCL:
   #Out_CIP_Req := #AlwaysON AND #State."CIP Tank";
   #Out_CIP_Line_Open := #AlwaysON AND #State."CIP Tank" AND #IN_FBAV_CIP AND #IN_FBAV_Outlet;
END_REGION

REGION Network 16: AV Outlet
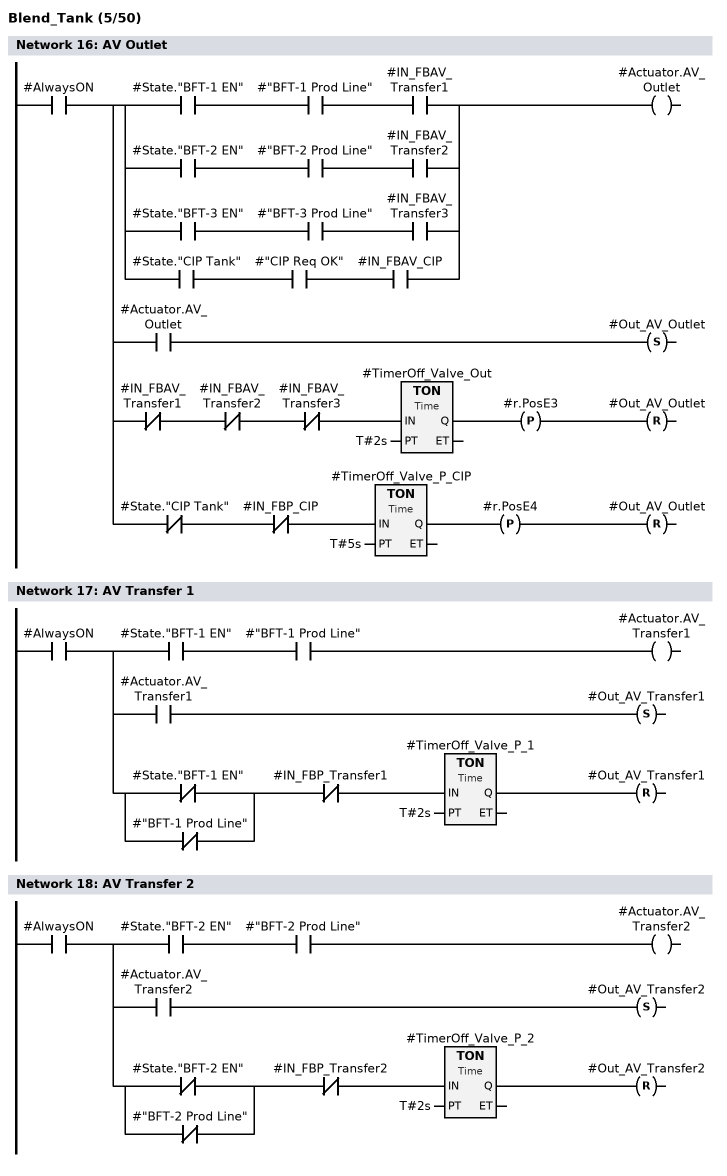
   RUNG wire#powerrail
      Contact( #AlwaysON )
      wire#w1
      Contact( #State."BFT-1 EN" )
      Contact( #"BFT-1 Prod Line" )
      Contact( #IN_FBAV_Transfer1 )
      wire#w2
      Coil( #Actuator.AV_Outlet )
   END_RUNG
   RUNG wire#w1
      Contact( #State."BFT-2 EN" )
      Contact( #"BFT-2 Prod Line" )
      Contact( #IN_FBAV_Transfer2 )
   END_RUNG wire#w2
   RUNG wire#w1
      Contact( #State."BFT-3 EN" )
      Contact( #"BFT-3 Prod Line" )
      Contact( #IN_FBAV_Transfer3 )
   END_RUNG wire#w2
   RUNG wire#w1
      Contact( #State."CIP Tank" )
      Contact( #"CIP Req OK" )
      Contact( #IN_FBAV_CIP )
   END_RUNG wire#w2
   RUNG wire#w1
      Contact( #Actuator.AV_Outlet )
      S_Coil( #Out_AV_Outlet )
   END_RUNG
   RUNG wire#w1
      I_Contact( #IN_FBAV_Transfer1 )
      I_Contact( #IN_FBAV_Transfer2 )
      I_Contact( #IN_FBAV_Transfer3 )
      { S7_Templates := "time_type := Time" } #TimerOff_Valve_Out.TON(pt := T#2s, et =>)
      P_Trig( #r.PosE3 )
      R_Coil( #Out_AV_Outlet )
   END_RUNG
   RUNG wire#w1
      I_Contact( #State."CIP Tank" )
      I_Contact( #IN_FBP_CIP )
      { S7_Templates := "time_type := Time" } #TimerOff_Valve_P_CIP.TON(pt := T#5s, et =>)
      P_Trig( #r.PosE4 )
      R_Coil( #Out_AV_Outlet )
   END_RUNG
   // the same network as SCL:
   #Actuator.AV_Outlet := #AlwaysON AND ((#State."BFT-1 EN" AND #"BFT-1 Prod Line" AND #IN_FBAV_Transfer1) OR (#State."BFT-2 EN" AND #"BFT-2 Prod Line" AND #IN_FBAV_Transfer2) OR (#State."BFT-3 EN" AND #"BFT-3 Prod Line" AND #IN_FBAV_Transfer3) OR (#State."CIP Tank" AND #"CIP Req OK" AND #IN_FBAV_CIP));
   IF #AlwaysON AND #Actuator.AV_Outlet THEN #Out_AV_Outlet := TRUE; END_IF;
   #TimerOff_Valve_Out(IN := #AlwaysON AND NOT #IN_FBAV_Transfer1 AND NOT #IN_FBAV_Transfer2 AND NOT #IN_FBAV_Transfer3,   // TON
                       PT := T#2s);
   #_w1 := #TimerOff_Valve_Out.Q AND NOT #r.PosE3;   // rising edge
   #r.PosE3 := #TimerOff_Valve_Out.Q;
   IF #_w1 THEN #Out_AV_Outlet := FALSE; END_IF;
   #TimerOff_Valve_P_CIP(IN := #AlwaysON AND NOT #State."CIP Tank" AND NOT #IN_FBP_CIP, PT := T#5s);   // TON
   #_w2 := #TimerOff_Valve_P_CIP.Q AND NOT #r.PosE4;   // rising edge
   #r.PosE4 := #TimerOff_Valve_P_CIP.Q;
   IF #_w2 THEN #Out_AV_Outlet := FALSE; END_IF;
END_REGION

REGION Network 17: AV Transfer 1
   RUNG wire#powerrail
      Contact( #AlwaysON )
      wire#w1
      Contact( #State."BFT-1 EN" )
      Contact( #"BFT-1 Prod Line" )
      Coil( #Actuator.AV_Transfer1 )
   END_RUNG
   RUNG wire#w1
      Contact( #Actuator.AV_Transfer1 )
      S_Coil( #Out_AV_Transfer1 )
   END_RUNG
   RUNG wire#w1
      I_Contact( #State."BFT-1 EN" )
      wire#w2
      I_Contact( #IN_FBP_Transfer1 )
      { S7_Templates := "time_type := Time" } #TimerOff_Valve_P_1.TON(pt := T#2s, et =>)
      R_Coil( #Out_AV_Transfer1 )
   END_RUNG
   RUNG wire#w1
      I_Contact( #"BFT-1 Prod Line" )
   END_RUNG wire#w2
   // the same network as SCL:
   #Actuator.AV_Transfer1 := #AlwaysON AND #State."BFT-1 EN" AND #"BFT-1 Prod Line";
   IF #AlwaysON AND #Actuator.AV_Transfer1 THEN #Out_AV_Transfer1 := TRUE; END_IF;
   #TimerOff_Valve_P_1(IN := #AlwaysON AND (NOT #State."BFT-1 EN" OR NOT #"BFT-1 Prod Line") AND NOT #IN_FBP_Transfer1,   // TON
                       PT := T#2s);
   IF #TimerOff_Valve_P_1.Q THEN #Out_AV_Transfer1 := FALSE; END_IF;
END_REGION

REGION Network 18: AV Transfer 2
   RUNG wire#powerrail
      Contact( #AlwaysON )
      wire#w1
      Contact( #State."BFT-2 EN" )
      Contact( #"BFT-2 Prod Line" )
      Coil( #Actuator.AV_Transfer2 )
   END_RUNG
   RUNG wire#w1
      Contact( #Actuator.AV_Transfer2 )
      S_Coil( #Out_AV_Transfer2 )
   END_RUNG
   RUNG wire#w1
      I_Contact( #State."BFT-2 EN" )
      wire#w2
      I_Contact( #IN_FBP_Transfer2 )
      { S7_Templates := "time_type := Time" } #TimerOff_Valve_P_2.TON(pt := T#2s, et =>)
      R_Coil( #Out_AV_Transfer2 )
   END_RUNG
   RUNG wire#w1
      I_Contact( #"BFT-2 Prod Line" )
   END_RUNG wire#w2
   // the same network as SCL:
   #Actuator.AV_Transfer2 := #AlwaysON AND #State."BFT-2 EN" AND #"BFT-2 Prod Line";
   IF #AlwaysON AND #Actuator.AV_Transfer2 THEN #Out_AV_Transfer2 := TRUE; END_IF;
   #TimerOff_Valve_P_2(IN := #AlwaysON AND (NOT #State."BFT-2 EN" OR NOT #"BFT-2 Prod Line") AND NOT #IN_FBP_Transfer2,   // TON
                       PT := T#2s);
   IF #TimerOff_Valve_P_2.Q THEN #Out_AV_Transfer2 := FALSE; END_IF;
END_REGION

REGION Network 19: AV Transfer 3
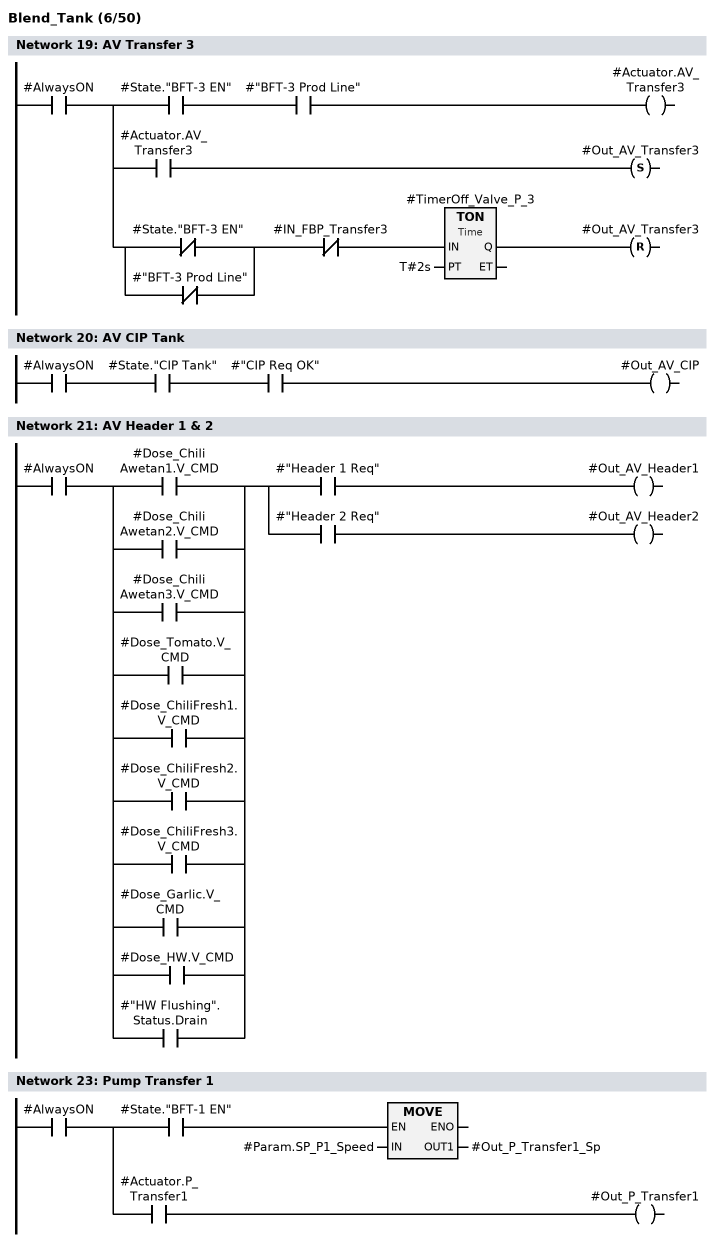
   RUNG wire#powerrail
      Contact( #AlwaysON )
      wire#w1
      Contact( #State."BFT-3 EN" )
      Contact( #"BFT-3 Prod Line" )
      Coil( #Actuator.AV_Transfer3 )
   END_RUNG
   RUNG wire#w1
      Contact( #Actuator.AV_Transfer3 )
      S_Coil( #Out_AV_Transfer3 )
   END_RUNG
   RUNG wire#w1
      I_Contact( #State."BFT-3 EN" )
      wire#w2
      I_Contact( #IN_FBP_Transfer3 )
      { S7_Templates := "time_type := Time" } #TimerOff_Valve_P_3.TON(pt := T#2s, et =>)
      R_Coil( #Out_AV_Transfer3 )
   END_RUNG
   RUNG wire#w1
      I_Contact( #"BFT-3 Prod Line" )
   END_RUNG wire#w2
   // the same network as SCL:
   #Actuator.AV_Transfer3 := #AlwaysON AND #State."BFT-3 EN" AND #"BFT-3 Prod Line";
   IF #AlwaysON AND #Actuator.AV_Transfer3 THEN #Out_AV_Transfer3 := TRUE; END_IF;
   #TimerOff_Valve_P_3(IN := #AlwaysON AND (NOT #State."BFT-3 EN" OR NOT #"BFT-3 Prod Line") AND NOT #IN_FBP_Transfer3,   // TON
                       PT := T#2s);
   IF #TimerOff_Valve_P_3.Q THEN #Out_AV_Transfer3 := FALSE; END_IF;
END_REGION

REGION Network 20: AV CIP Tank
   RUNG wire#powerrail
      Contact( #AlwaysON )
      Contact( #State."CIP Tank" )
      Contact( #"CIP Req OK" )
      Coil( #Out_AV_CIP )
   END_RUNG
   // the same network as SCL:
   #Out_AV_CIP := #AlwaysON AND #State."CIP Tank" AND #"CIP Req OK";
END_REGION

REGION Network 21: AV Header 1 & 2
   RUNG wire#powerrail
      Contact( #AlwaysON )
      wire#w1
      Contact( #Dose_ChiliAwetan1.V_CMD )
      wire#w2
      Contact( #"Header 1 Req" )
      Coil( #Out_AV_Header1 )
   END_RUNG
   RUNG wire#w1
      Contact( #Dose_ChiliAwetan2.V_CMD )
   END_RUNG wire#w2
   RUNG wire#w1
      Contact( #Dose_ChiliAwetan3.V_CMD )
   END_RUNG wire#w2
   RUNG wire#w1
      Contact( #Dose_Tomato.V_CMD )
   END_RUNG wire#w2
   RUNG wire#w1
      Contact( #Dose_ChiliFresh1.V_CMD )
   END_RUNG wire#w2
   RUNG wire#w1
      Contact( #Dose_ChiliFresh2.V_CMD )
   END_RUNG wire#w2
   RUNG wire#w1
      Contact( #Dose_ChiliFresh3.V_CMD )
   END_RUNG wire#w2
   RUNG wire#w1
      Contact( #Dose_Garlic.V_CMD )
   END_RUNG wire#w2
   RUNG wire#w1
      Contact( #Dose_HW.V_CMD )
   END_RUNG wire#w2
   RUNG wire#w1
      Contact( #"HW Flushing".Status.Drain )
   END_RUNG wire#w2
   RUNG wire#w2
      Contact( #"Header 2 Req" )
      Coil( #Out_AV_Header2 )
   END_RUNG
   // the same network as SCL:
   #_w1 := #AlwaysON AND (#Dose_ChiliAwetan1.V_CMD OR #Dose_ChiliAwetan2.V_CMD OR #Dose_ChiliAwetan3.V_CMD OR #Dose_Tomato.V_CMD OR #Dose_ChiliFresh1.V_CMD OR #Dose_ChiliFresh2.V_CMD OR #Dose_ChiliFresh3.V_CMD OR #Dose_Garlic.V_CMD OR #Dose_HW.V_CMD OR #"HW Flushing".Status.Drain);
   #Out_AV_Header1 := #_w1 AND #"Header 1 Req";
   #Out_AV_Header2 := #_w1 AND #"Header 2 Req";
END_REGION

REGION Network 23: Pump Transfer 1
   RUNG wire#powerrail
      Contact( #AlwaysON )
      wire#w1
      Contact( #State."BFT-1 EN" )
      Move(in := #Param.SP_P1_Speed, out1 => #Out_P_Transfer1_Sp)
   END_RUNG
   RUNG wire#w1
      Contact( #Actuator.P_Transfer1 )
      Coil( #Out_P_Transfer1 )
   END_RUNG
   // the same network as SCL:
   IF #AlwaysON AND #State."BFT-1 EN" THEN #Out_P_Transfer1_Sp := #Param.SP_P1_Speed; END_IF;
   #Out_P_Transfer1 := #AlwaysON AND #Actuator.P_Transfer1;
END_REGION

REGION Network 24: Pump Transfer 2
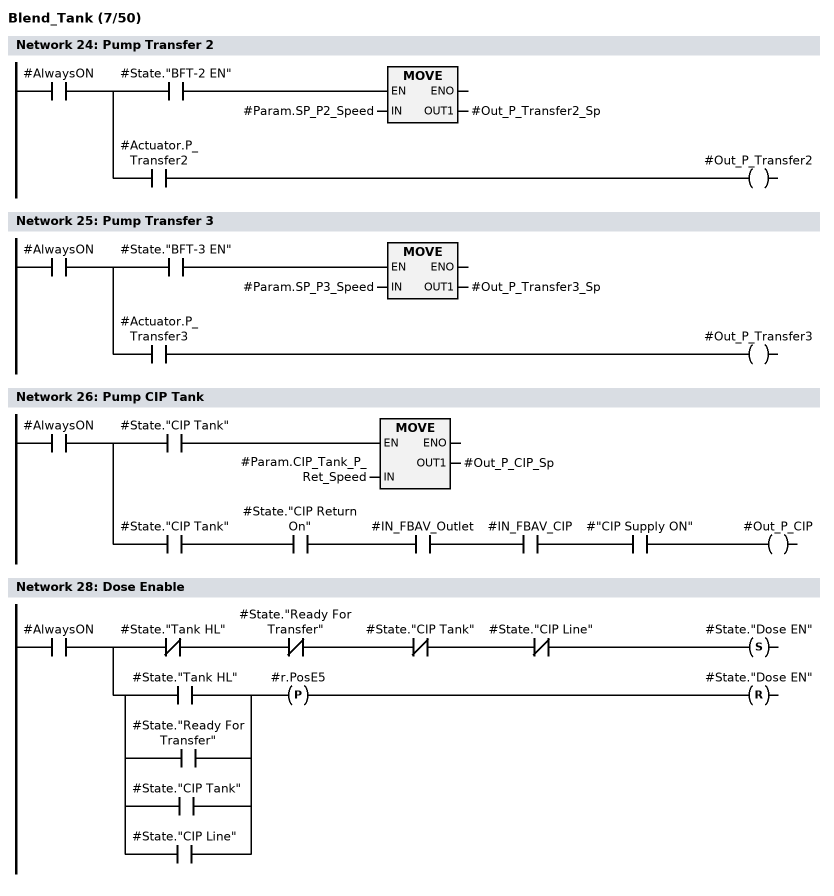
   RUNG wire#powerrail
      Contact( #AlwaysON )
      wire#w1
      Contact( #State."BFT-2 EN" )
      Move(in := #Param.SP_P2_Speed, out1 => #Out_P_Transfer2_Sp)
   END_RUNG
   RUNG wire#w1
      Contact( #Actuator.P_Transfer2 )
      Coil( #Out_P_Transfer2 )
   END_RUNG
   // the same network as SCL:
   IF #AlwaysON AND #State."BFT-2 EN" THEN #Out_P_Transfer2_Sp := #Param.SP_P2_Speed; END_IF;
   #Out_P_Transfer2 := #AlwaysON AND #Actuator.P_Transfer2;
END_REGION

REGION Network 25: Pump Transfer 3
   RUNG wire#powerrail
      Contact( #AlwaysON )
      wire#w1
      Contact( #State."BFT-3 EN" )
      Move(in := #Param.SP_P3_Speed, out1 => #Out_P_Transfer3_Sp)
   END_RUNG
   RUNG wire#w1
      Contact( #Actuator.P_Transfer3 )
      Coil( #Out_P_Transfer3 )
   END_RUNG
   // the same network as SCL:
   IF #AlwaysON AND #State."BFT-3 EN" THEN #Out_P_Transfer3_Sp := #Param.SP_P3_Speed; END_IF;
   #Out_P_Transfer3 := #AlwaysON AND #Actuator.P_Transfer3;
END_REGION

REGION Network 26: Pump CIP Tank
   RUNG wire#powerrail
      Contact( #AlwaysON )
      wire#w1
      Contact( #State."CIP Tank" )
      Move(in := #Param.CIP_Tank_P_Ret_Speed, out1 => #Out_P_CIP_Sp)
   END_RUNG
   RUNG wire#w1
      Contact( #State."CIP Tank" )
      Contact( #State."CIP Return On" )
      Contact( #IN_FBAV_Outlet )
      Contact( #IN_FBAV_CIP )
      Contact( #"CIP Supply ON" )
      Coil( #Out_P_CIP )
   END_RUNG
   // the same network as SCL:
   IF #AlwaysON AND #State."CIP Tank" THEN #Out_P_CIP_Sp := #Param.CIP_Tank_P_Ret_Speed; END_IF;
   #Out_P_CIP := #AlwaysON AND #State."CIP Tank" AND #State."CIP Return On" AND #IN_FBAV_Outlet AND #IN_FBAV_CIP AND #"CIP Supply ON";
END_REGION

REGION Network 28: Dose Enable
   RUNG wire#powerrail
      Contact( #AlwaysON )
      wire#w1
      I_Contact( #State."Tank HL" )
      I_Contact( #State."Ready For Transfer" )
      I_Contact( #State."CIP Tank" )
      I_Contact( #State."CIP Line" )
      S_Coil( #State."Dose EN" )
   END_RUNG
   RUNG wire#w1
      Contact( #State."Tank HL" )
      wire#w2
      P_Trig( #r.PosE5 )
      R_Coil( #State."Dose EN" )
   END_RUNG
   RUNG wire#w1
      Contact( #State."Ready For Transfer" )
   END_RUNG wire#w2
   RUNG wire#w1
      Contact( #State."CIP Tank" )
   END_RUNG wire#w2
   RUNG wire#w1
      Contact( #State."CIP Line" )
   END_RUNG wire#w2
   // the same network as SCL:
   IF #AlwaysON AND NOT #State."Tank HL" AND NOT #State."Ready For Transfer" AND NOT #State."CIP Tank" AND NOT #State."CIP Line" THEN
       #State."Dose EN" := TRUE;
   END_IF;
   #_w1 := #AlwaysON AND (#State."Tank HL" OR #State."Ready For Transfer" OR #State."CIP Tank" OR #State."CIP Line");
   #_w2 := #_w1 AND NOT #r.PosE5;   // rising edge
   #r.PosE5 := #_w1;
   IF #_w2 THEN #State."Dose EN" := FALSE; END_IF;
END_REGION

NETWORK
TITLE = Raw Material & Tank Dose State
// Raw Material Dose State
      O     #Dose_ChiliAwetan1.QDOSERun;
      O     #Dose_ChiliAwetan2.QDOSERun;
      O     #Dose_ChiliAwetan3.QDOSERun;
      O     #Dose_Tomato.QDOSERun;
      O     #Dose_ChiliFresh1.QDOSERun;
      O     #Dose_ChiliFresh2.QDOSERun;
      O     #Dose_ChiliFresh3.QDOSERun;
      O     #Dose_Garlic.QDOSERun;
      O     #Dose_HW.QDOSERun;
      =     #State."RM Dose";

// Dose Run State
      O     #State."RM Dose";
      O     #Dose_Vinegar.QDOSERun;
      O     #Dose_Sugar.QDOSERun;
      O     #Dose_Salt.QDOSERun;
      O     #Dose_ProWater.QDOSERun;
      O     #Dose_Homomixer.QDOSERun;
      =     #State."Dose On Prog";


REGION Network 31: Header 1 & 2 --- Vinegar --- Sugar --- Salt --- ProWater --- Homomixer Enable
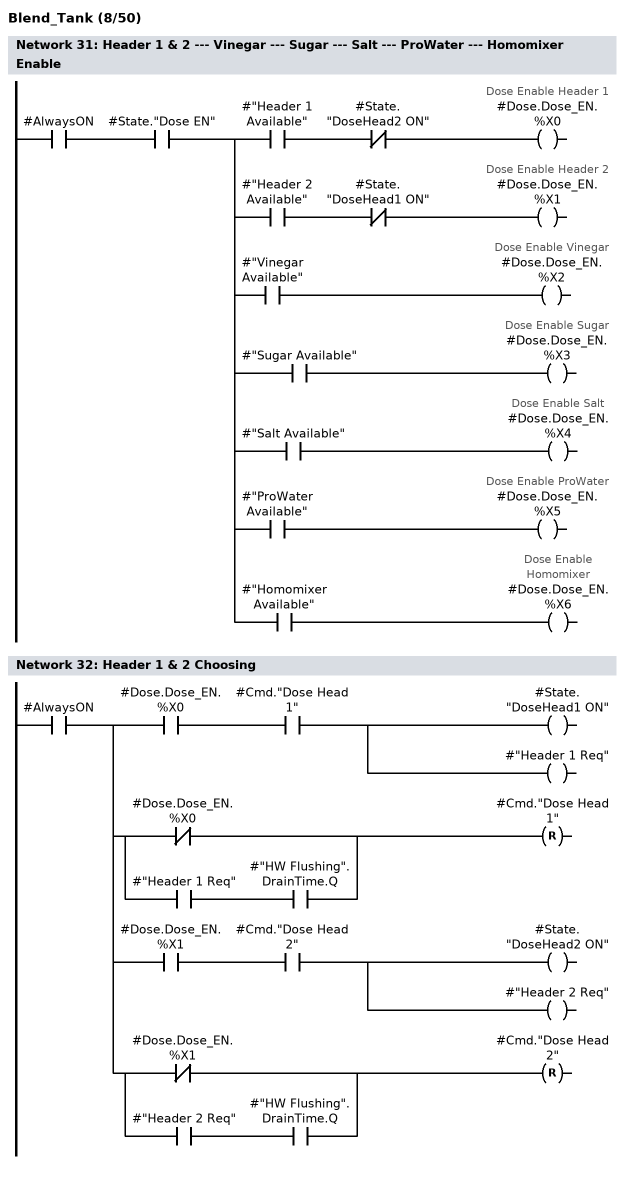
   RUNG wire#powerrail
      Contact( #AlwaysON )
      Contact( #State."Dose EN" )
      wire#w1
      Contact( #"Header 1 Available" )
      I_Contact( #State."DoseHead2 ON" )
      Coil( #Dose.Dose_EN.%X0 )   // Dose Enable Header 1
   END_RUNG
   RUNG wire#w1
      Contact( #"Header 2 Available" )
      I_Contact( #State."DoseHead1 ON" )
      Coil( #Dose.Dose_EN.%X1 )   // Dose Enable Header 2
   END_RUNG
   RUNG wire#w1
      Contact( #"Vinegar Available" )
      Coil( #Dose.Dose_EN.%X2 )   // Dose Enable Vinegar
   END_RUNG
   RUNG wire#w1
      Contact( #"Sugar Available" )
      Coil( #Dose.Dose_EN.%X3 )   // Dose Enable Sugar
   END_RUNG
   RUNG wire#w1
      Contact( #"Salt Available" )
      Coil( #Dose.Dose_EN.%X4 )   // Dose Enable Salt
   END_RUNG
   RUNG wire#w1
      Contact( #"ProWater Available" )
      Coil( #Dose.Dose_EN.%X5 )   // Dose Enable ProWater
   END_RUNG
   RUNG wire#w1
      Contact( #"Homomixer Available" )
      Coil( #Dose.Dose_EN.%X6 )   // Dose Enable Homomixer
   END_RUNG
   // the same network as SCL:
   #_w1 := #AlwaysON AND #State."Dose EN";
   #Dose.Dose_EN.%X0 := #_w1 AND #"Header 1 Available" AND NOT #State."DoseHead2 ON";   // Dose Enable Header 1
   #Dose.Dose_EN.%X1 := #_w1 AND #"Header 2 Available" AND NOT #State."DoseHead1 ON";   // Dose Enable Header 2
   #Dose.Dose_EN.%X2 := #_w1 AND #"Vinegar Available";   // Dose Enable Vinegar
   #Dose.Dose_EN.%X3 := #_w1 AND #"Sugar Available";   // Dose Enable Sugar
   #Dose.Dose_EN.%X4 := #_w1 AND #"Salt Available";   // Dose Enable Salt
   #Dose.Dose_EN.%X5 := #_w1 AND #"ProWater Available";   // Dose Enable ProWater
   #Dose.Dose_EN.%X6 := #_w1 AND #"Homomixer Available";   // Dose Enable Homomixer
END_REGION

REGION Network 32: Header 1 & 2 Choosing
   RUNG wire#powerrail
      Contact( #AlwaysON )
      wire#w1
      Contact( #Dose.Dose_EN.%X0 )
      Contact( #Cmd."Dose Head 1" )
      wire#w2
      Coil( #State."DoseHead1 ON" )
   END_RUNG
   RUNG wire#w2
      Coil( #"Header 1 Req" )
   END_RUNG
   RUNG wire#w1
      I_Contact( #Dose.Dose_EN.%X0 )
      wire#w3
      R_Coil( #Cmd."Dose Head 1" )
   END_RUNG
   RUNG wire#w1
      Contact( #"Header 1 Req" )
      Contact( #"HW Flushing".DrainTime.Q )
   END_RUNG wire#w3
   RUNG wire#w1
      Contact( #Dose.Dose_EN.%X1 )
      Contact( #Cmd."Dose Head 2" )
      wire#w4
      Coil( #State."DoseHead2 ON" )
   END_RUNG
   RUNG wire#w4
      Coil( #"Header 2 Req" )
   END_RUNG
   RUNG wire#w1
      I_Contact( #Dose.Dose_EN.%X1 )
      wire#w5
      R_Coil( #Cmd."Dose Head 2" )
   END_RUNG
   RUNG wire#w1
      Contact( #"Header 2 Req" )
      Contact( #"HW Flushing".DrainTime.Q )
   END_RUNG wire#w5
   // the same network as SCL:
   #State."DoseHead1 ON" := #AlwaysON AND #Dose.Dose_EN.%X0 AND #Cmd."Dose Head 1";
   #"Header 1 Req" := #State."DoseHead1 ON";
   IF #AlwaysON AND (NOT #Dose.Dose_EN.%X0 OR (#"Header 1 Req" AND #"HW Flushing".DrainTime.Q)) THEN
       #Cmd."Dose Head 1" := FALSE;
   END_IF;
   #State."DoseHead2 ON" := #AlwaysON AND #Dose.Dose_EN.%X1 AND #Cmd."Dose Head 2";
   #"Header 2 Req" := #State."DoseHead2 ON";
   IF #AlwaysON AND (NOT #Dose.Dose_EN.%X1 OR (#"Header 2 Req" AND #"HW Flushing".DrainTime.Q)) THEN
       #Cmd."Dose Head 2" := FALSE;
   END_IF;
END_REGION

NETWORK
TITLE = Header 1 & 2 Request
// Header 1 Request
//      O     #Dose.Dose_Header_Req.%X0// ChiliAwetan1 Header1 Req
//      O     #Dose.Dose_Header_Req.%X1// ChiliAwetan2 Header1 Req
//      O     #Dose.Dose_Header_Req.%X2// ChiliAwetan3 Header1 Req
//      O     #Dose.Dose_Header_Req.%X3// Tomato Header1 Req
//      O     #Dose.Dose_Header_Req.%X4// ChiliFresh1 Header1 Req
//      O     #Dose.Dose_Header_Req.%X5// ChiliFresh2 Header1 Req
//      O     #Dose.Dose_Header_Req.%X6// ChiliFresh3 Header1 Req
//      O     #Dose.Dose_Header_Req.%X7// Garlic Header1 Req
//      O     #Dose.Dose_Header_Req.%X8// HotWater Header1 Req
//     =     #"Header 1 Req"

// Header 2 Request
//      O     #Dose.Dose_Header_Req.%X16// ChiliAwetan1 Header2 Req
//      O     #Dose.Dose_Header_Req.%X17// ChiliAwetan2 Header2 Req
//      O     #Dose.Dose_Header_Req.%X18// ChiliAwetan3 Header2 Req
//      O     #Dose.Dose_Header_Req.%X19// Tomato Header2 Req
//      O     #Dose.Dose_Header_Req.%X20// ChiliFresh1 Header2 Req
//      O     #Dose.Dose_Header_Req.%X21// ChiliFresh2 Header2 Req
//      O     #Dose.Dose_Header_Req.%X22// ChiliFresh3 Header2 Req
//      O     #Dose.Dose_Header_Req.%X23// Garlic Header2 Req
//      O     #Dose.Dose_Header_Req.%X24// HotWater Header2 Req
//      =     #"Header 2 Req"


REGION Network 36: ChiliAwetan1 Setpoint
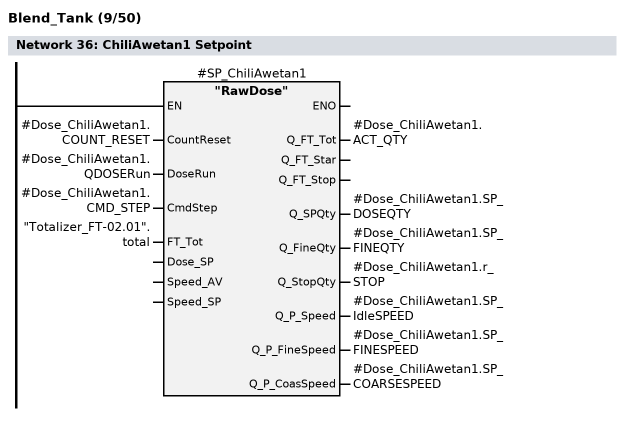
   RUNG wire#powerrail
      #SP_ChiliAwetan1(CountReset := #Dose_ChiliAwetan1.COUNT_RESET, DoseRun := #Dose_ChiliAwetan1.QDOSERun, CmdStep := #Dose_ChiliAwetan1.CMD_STEP, FT_Tot := "Totalizer_FT-02.01".total, Dose_SP :=, Speed_AV :=, Speed_SP :=, Q_FT_Tot => #Dose_ChiliAwetan1.ACT_QTY, Q_FT_Star =>, Q_FT_Stop =>, Q_SPQty => #Dose_ChiliAwetan1.SP_DOSEQTY, Q_FineQty => #Dose_ChiliAwetan1.SP_FINEQTY, Q_StopQty => #Dose_ChiliAwetan1.r_STOP, Q_P_Speed => #Dose_ChiliAwetan1.SP_IdleSPEED, Q_P_FineSpeed => #Dose_ChiliAwetan1.SP_FINESPEED, Q_P_CoasSpeed => #Dose_ChiliAwetan1.SP_COARSESPEED)
   END_RUNG
   // the same network as SCL:
   #SP_ChiliAwetan1(CountReset := #Dose_ChiliAwetan1.COUNT_RESET,   // "RawDose"
                    DoseRun := #Dose_ChiliAwetan1.QDOSERun,
                    CmdStep := #Dose_ChiliAwetan1.CMD_STEP,
                    FT_Tot := "Totalizer_FT-02.01".total,
                    Q_FT_Tot => #Dose_ChiliAwetan1.ACT_QTY,
                    Q_SPQty => #Dose_ChiliAwetan1.SP_DOSEQTY,
                    Q_FineQty => #Dose_ChiliAwetan1.SP_FINEQTY,
                    Q_StopQty => #Dose_ChiliAwetan1.r_STOP,
                    Q_P_Speed => #Dose_ChiliAwetan1.SP_IdleSPEED,
                    Q_P_FineSpeed => #Dose_ChiliAwetan1.SP_FINESPEED,
                    Q_P_CoasSpeed => #Dose_ChiliAwetan1.SP_COARSESPEED);
END_REGION

REGION Network 37: Command Dose ChiliAwetan1
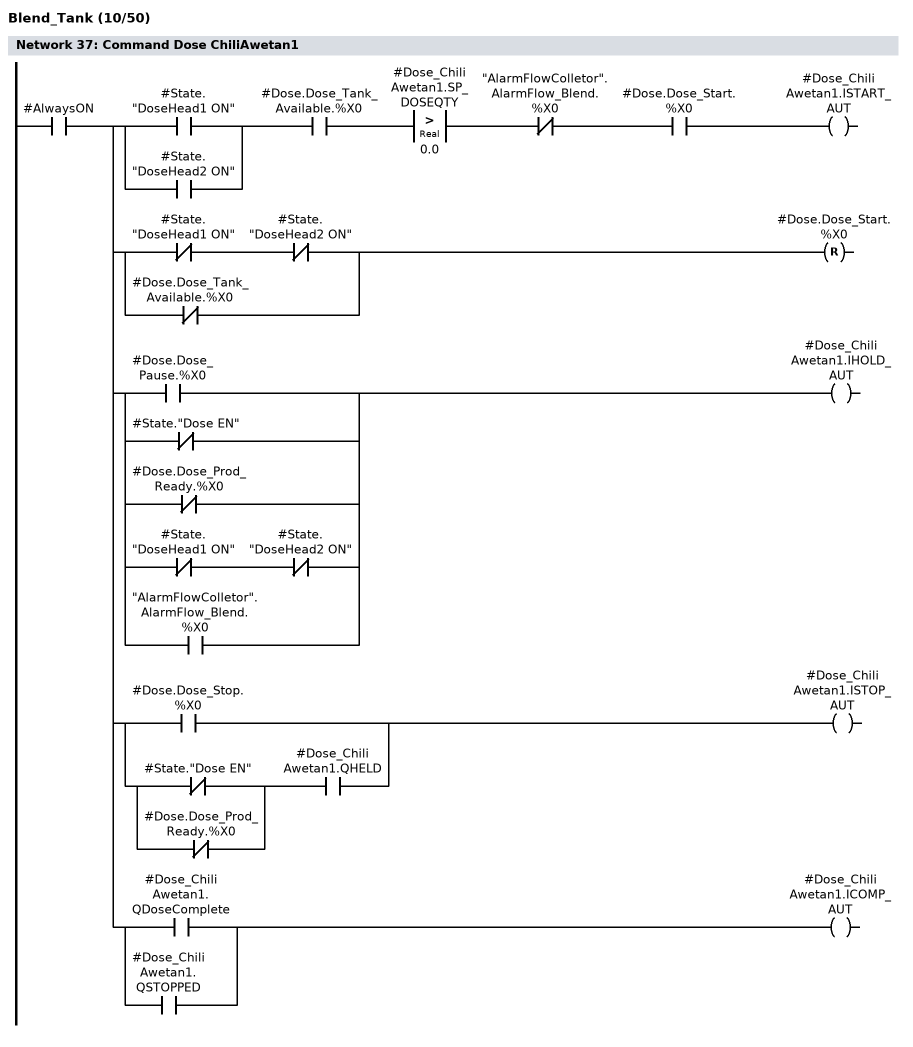
   RUNG wire#powerrail
      Contact( #AlwaysON )
      wire#w1
      Contact( #State."DoseHead1 ON" )
      wire#w2
      Contact( #Dose.Dose_Tank_Available.%X0 )
      { S7_Templates := "SrcType := Real" } GT_Contact(in1 := #Dose_ChiliAwetan1.SP_DOSEQTY, in2 := 0.0)
      I_Contact( "AlarmFlowColletor".AlarmFlow_Blend.%X0 )
      Contact( #Dose.Dose_Start.%X0 )
      Coil( #Dose_ChiliAwetan1.ISTART_AUT )
   END_RUNG
   RUNG wire#w1
      Contact( #State."DoseHead2 ON" )
   END_RUNG wire#w2
   RUNG wire#w1
      I_Contact( #State."DoseHead1 ON" )
      I_Contact( #State."DoseHead2 ON" )
      wire#w3
      R_Coil( #Dose.Dose_Start.%X0 )
   END_RUNG
   RUNG wire#w1
      I_Contact( #Dose.Dose_Tank_Available.%X0 )
   END_RUNG wire#w3
   RUNG wire#w1
      Contact( #Dose.Dose_Pause.%X0 )
      wire#w4
      Coil( #Dose_ChiliAwetan1.IHOLD_AUT )
   END_RUNG
   RUNG wire#w1
      I_Contact( #State."Dose EN" )
   END_RUNG wire#w4
   RUNG wire#w1
      I_Contact( #Dose.Dose_Prod_Ready.%X0 )
   END_RUNG wire#w4
   RUNG wire#w1
      I_Contact( #State."DoseHead1 ON" )
      I_Contact( #State."DoseHead2 ON" )
   END_RUNG wire#w4
   RUNG wire#w1
      Contact( "AlarmFlowColletor".AlarmFlow_Blend.%X0 )
   END_RUNG wire#w4
   RUNG wire#w1
      Contact( #Dose.Dose_Stop.%X0 )
      wire#w5
      Coil( #Dose_ChiliAwetan1.ISTOP_AUT )
   END_RUNG
   RUNG wire#w1
      I_Contact( #State."Dose EN" )
      wire#w6
      Contact( #Dose_ChiliAwetan1.QHELD )
   END_RUNG wire#w5
   RUNG wire#w1
      I_Contact( #Dose.Dose_Prod_Ready.%X0 )
   END_RUNG wire#w6
   RUNG wire#w1
      Contact( #Dose_ChiliAwetan1.QDoseComplete )
      wire#w7
      Coil( #Dose_ChiliAwetan1.ICOMP_AUT )
   END_RUNG
   RUNG wire#w1
      Contact( #Dose_ChiliAwetan1.QSTOPPED )
   END_RUNG wire#w7
   // the same network as SCL:
   #Dose_ChiliAwetan1.ISTART_AUT := #AlwaysON AND (#State."DoseHead1 ON" OR #State."DoseHead2 ON") AND #Dose.Dose_Tank_Available.%X0 AND (#Dose_ChiliAwetan1.SP_DOSEQTY > 0.0) AND NOT "AlarmFlowColletor".AlarmFlow_Blend.%X0 AND #Dose.Dose_Start.%X0;
   IF #AlwaysON AND ((NOT #State."DoseHead1 ON" AND NOT #State."DoseHead2 ON") OR NOT #Dose.Dose_Tank_Available.%X0) THEN
       #Dose.Dose_Start.%X0 := FALSE;
   END_IF;
   #Dose_ChiliAwetan1.IHOLD_AUT := #AlwaysON AND (#Dose.Dose_Pause.%X0 OR NOT #State."Dose EN" OR NOT #Dose.Dose_Prod_Ready.%X0 OR (NOT #State."DoseHead1 ON" AND NOT #State."DoseHead2 ON") OR "AlarmFlowColletor".AlarmFlow_Blend.%X0);
   #Dose_ChiliAwetan1.ISTOP_AUT := #AlwaysON AND (#Dose.Dose_Stop.%X0 OR ((NOT #State."Dose EN" OR NOT #Dose.Dose_Prod_Ready.%X0) AND #Dose_ChiliAwetan1.QHELD));
   #Dose_ChiliAwetan1.ICOMP_AUT := #AlwaysON AND (#Dose_ChiliAwetan1.QDoseComplete OR #Dose_ChiliAwetan1.QSTOPPED);
END_REGION

REGION Network 38: Dose ChiliAwetan1
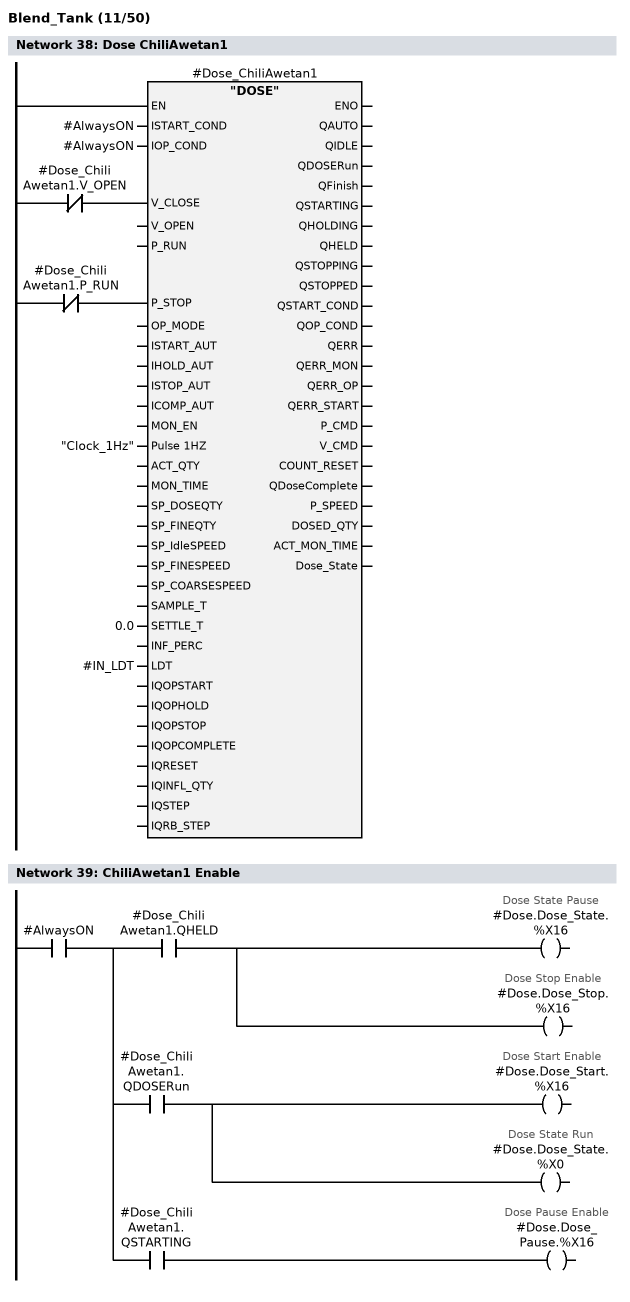
   RUNG wire#powerrail
      #Dose_ChiliAwetan1(V_CLOSE := wire#w1, P_STOP := wire#w2, ISTART_COND := #AlwaysON, IOP_COND := #AlwaysON, V_OPEN :=, P_RUN :=, OP_MODE :=, ISTART_AUT :=, IHOLD_AUT :=, ISTOP_AUT :=, ICOMP_AUT :=, MON_EN :=, "Pulse 1HZ" := "Clock_1Hz", ACT_QTY :=, MON_TIME :=, SP_DOSEQTY :=, SP_FINEQTY :=, SP_IdleSPEED :=, SP_FINESPEED :=, SP_COARSESPEED :=, SAMPLE_T :=, SETTLE_T := 0.0, INF_PERC :=, LDT := #IN_LDT, IQOPSTART :=, IQOPHOLD :=, IQOPSTOP :=, IQOPCOMPLETE :=, IQRESET :=, IQINFL_QTY :=, IQSTEP :=, IQRB_STEP :=, QAUTO =>, QIDLE =>, QDOSERun =>, QFinish =>, QSTARTING =>, QHOLDING =>, QHELD =>, QSTOPPING =>, QSTOPPED =>, QSTART_COND =>, QOP_COND =>, QERR =>, QERR_MON =>, QERR_OP =>, QERR_START =>, P_CMD =>, V_CMD =>, COUNT_RESET =>, QDoseComplete =>, P_SPEED =>, DOSED_QTY =>, ACT_MON_TIME =>, Dose_State =>)
   END_RUNG
   RUNG wire#powerrail
      I_Contact( #Dose_ChiliAwetan1.V_OPEN )
   END_RUNG wire#w1
   RUNG wire#powerrail
      I_Contact( #Dose_ChiliAwetan1.P_RUN )
   END_RUNG wire#w2
   // the same network as SCL:
   #Dose_ChiliAwetan1(ISTART_COND := #AlwaysON,   // "DOSE"
                      IOP_COND := #AlwaysON,
                      V_CLOSE := NOT #Dose_ChiliAwetan1.V_OPEN,
                      P_STOP := NOT #Dose_ChiliAwetan1.P_RUN,
                      "Pulse 1HZ" := "Clock_1Hz",
                      SETTLE_T := 0.0,
                      LDT := #IN_LDT);
END_REGION

REGION Network 39: ChiliAwetan1 Enable
   RUNG wire#powerrail
      Contact( #AlwaysON )
      wire#w1
      Contact( #Dose_ChiliAwetan1.QHELD )
      wire#w2
      Coil( #Dose.Dose_State.%X16 )   // Dose State Pause
   END_RUNG
   RUNG wire#w2
      Coil( #Dose.Dose_Stop.%X16 )   // Dose Stop Enable
   END_RUNG
   RUNG wire#w1
      Contact( #Dose_ChiliAwetan1.QDOSERun )
      wire#w3
      Coil( #Dose.Dose_Start.%X16 )   // Dose Start Enable
   END_RUNG
   RUNG wire#w3
      Coil( #Dose.Dose_State.%X0 )   // Dose State Run
   END_RUNG
   RUNG wire#w1
      Contact( #Dose_ChiliAwetan1.QSTARTING )
      Coil( #Dose.Dose_Pause.%X16 )   // Dose Pause Enable
   END_RUNG
   // the same network as SCL:
   #Dose.Dose_State.%X16 := #AlwaysON AND #Dose_ChiliAwetan1.QHELD;   // Dose State Pause
   #Dose.Dose_Stop.%X16 := #Dose.Dose_State.%X16;   // Dose Stop Enable
   #Dose.Dose_Start.%X16 := #AlwaysON AND #Dose_ChiliAwetan1.QDOSERun;   // Dose Start Enable
   #Dose.Dose_State.%X0 := #Dose.Dose_Start.%X16;   // Dose State Run
   #Dose.Dose_Pause.%X16 := #AlwaysON AND #Dose_ChiliAwetan1.QSTARTING;   // Dose Pause Enable
END_REGION

REGION Network 40: ChiliAwetan1 Header Req
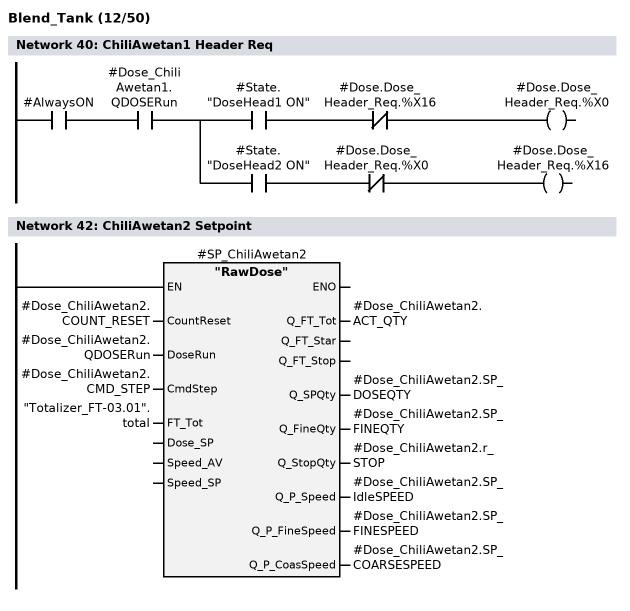
   RUNG wire#powerrail
      Contact( #AlwaysON )
      Contact( #Dose_ChiliAwetan1.QDOSERun )
      wire#w1
      Contact( #State."DoseHead1 ON" )
      I_Contact( #Dose.Dose_Header_Req.%X16 )
      Coil( #Dose.Dose_Header_Req.%X0 )
   END_RUNG
   RUNG wire#w1
      Contact( #State."DoseHead2 ON" )
      I_Contact( #Dose.Dose_Header_Req.%X0 )
      Coil( #Dose.Dose_Header_Req.%X16 )
   END_RUNG
   // the same network as SCL:
   #_w1 := #AlwaysON AND #Dose_ChiliAwetan1.QDOSERun;
   #Dose.Dose_Header_Req.%X0 := #_w1 AND #State."DoseHead1 ON" AND NOT #Dose.Dose_Header_Req.%X16;
   #Dose.Dose_Header_Req.%X16 := #_w1 AND #State."DoseHead2 ON" AND NOT #Dose.Dose_Header_Req.%X0;
END_REGION

REGION Network 42: ChiliAwetan2 Setpoint
   RUNG wire#powerrail
      #SP_ChiliAwetan2(CountReset := #Dose_ChiliAwetan2.COUNT_RESET, DoseRun := #Dose_ChiliAwetan2.QDOSERun, CmdStep := #Dose_ChiliAwetan2.CMD_STEP, FT_Tot := "Totalizer_FT-03.01".total, Dose_SP :=, Speed_AV :=, Speed_SP :=, Q_FT_Tot => #Dose_ChiliAwetan2.ACT_QTY, Q_FT_Star =>, Q_FT_Stop =>, Q_SPQty => #Dose_ChiliAwetan2.SP_DOSEQTY, Q_FineQty => #Dose_ChiliAwetan2.SP_FINEQTY, Q_StopQty => #Dose_ChiliAwetan2.r_STOP, Q_P_Speed => #Dose_ChiliAwetan2.SP_IdleSPEED, Q_P_FineSpeed => #Dose_ChiliAwetan2.SP_FINESPEED, Q_P_CoasSpeed => #Dose_ChiliAwetan2.SP_COARSESPEED)
   END_RUNG
   // the same network as SCL:
   #SP_ChiliAwetan2(CountReset := #Dose_ChiliAwetan2.COUNT_RESET,   // "RawDose"
                    DoseRun := #Dose_ChiliAwetan2.QDOSERun,
                    CmdStep := #Dose_ChiliAwetan2.CMD_STEP,
                    FT_Tot := "Totalizer_FT-03.01".total,
                    Q_FT_Tot => #Dose_ChiliAwetan2.ACT_QTY,
                    Q_SPQty => #Dose_ChiliAwetan2.SP_DOSEQTY,
                    Q_FineQty => #Dose_ChiliAwetan2.SP_FINEQTY,
                    Q_StopQty => #Dose_ChiliAwetan2.r_STOP,
                    Q_P_Speed => #Dose_ChiliAwetan2.SP_IdleSPEED,
                    Q_P_FineSpeed => #Dose_ChiliAwetan2.SP_FINESPEED,
                    Q_P_CoasSpeed => #Dose_ChiliAwetan2.SP_COARSESPEED);
END_REGION

REGION Network 43: Command Dose ChiliAwetan2
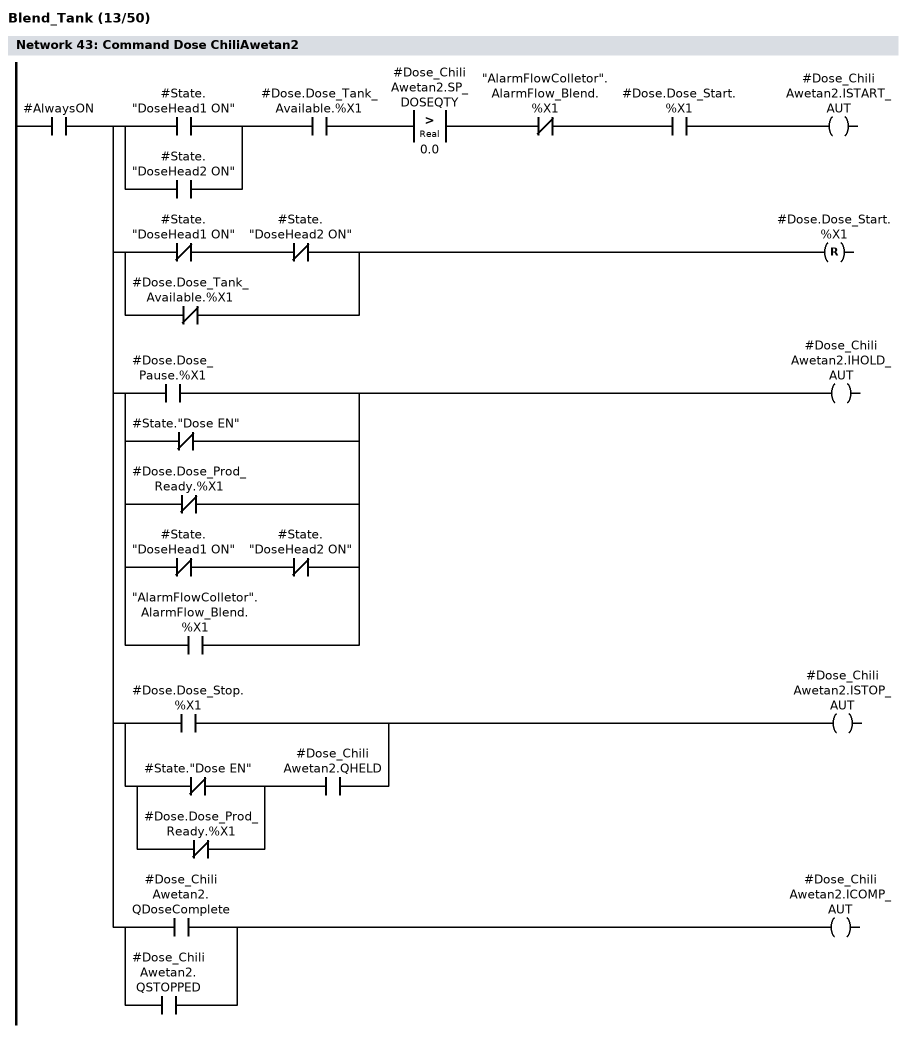
   RUNG wire#powerrail
      Contact( #AlwaysON )
      wire#w1
      Contact( #State."DoseHead1 ON" )
      wire#w2
      Contact( #Dose.Dose_Tank_Available.%X1 )
      { S7_Templates := "SrcType := Real" } GT_Contact(in1 := #Dose_ChiliAwetan2.SP_DOSEQTY, in2 := 0.0)
      I_Contact( "AlarmFlowColletor".AlarmFlow_Blend.%X1 )
      Contact( #Dose.Dose_Start.%X1 )
      Coil( #Dose_ChiliAwetan2.ISTART_AUT )
   END_RUNG
   RUNG wire#w1
      Contact( #State."DoseHead2 ON" )
   END_RUNG wire#w2
   RUNG wire#w1
      I_Contact( #State."DoseHead1 ON" )
      I_Contact( #State."DoseHead2 ON" )
      wire#w3
      R_Coil( #Dose.Dose_Start.%X1 )
   END_RUNG
   RUNG wire#w1
      I_Contact( #Dose.Dose_Tank_Available.%X1 )
   END_RUNG wire#w3
   RUNG wire#w1
      Contact( #Dose.Dose_Pause.%X1 )
      wire#w4
      Coil( #Dose_ChiliAwetan2.IHOLD_AUT )
   END_RUNG
   RUNG wire#w1
      I_Contact( #State."Dose EN" )
   END_RUNG wire#w4
   RUNG wire#w1
      I_Contact( #Dose.Dose_Prod_Ready.%X1 )
   END_RUNG wire#w4
   RUNG wire#w1
      I_Contact( #State."DoseHead1 ON" )
      I_Contact( #State."DoseHead2 ON" )
   END_RUNG wire#w4
   RUNG wire#w1
      Contact( "AlarmFlowColletor".AlarmFlow_Blend.%X1 )
   END_RUNG wire#w4
   RUNG wire#w1
      Contact( #Dose.Dose_Stop.%X1 )
      wire#w5
      Coil( #Dose_ChiliAwetan2.ISTOP_AUT )
   END_RUNG
   RUNG wire#w1
      I_Contact( #State."Dose EN" )
      wire#w6
      Contact( #Dose_ChiliAwetan2.QHELD )
   END_RUNG wire#w5
   RUNG wire#w1
      I_Contact( #Dose.Dose_Prod_Ready.%X1 )
   END_RUNG wire#w6
   RUNG wire#w1
      Contact( #Dose_ChiliAwetan2.QDoseComplete )
      wire#w7
      Coil( #Dose_ChiliAwetan2.ICOMP_AUT )
   END_RUNG
   RUNG wire#w1
      Contact( #Dose_ChiliAwetan2.QSTOPPED )
   END_RUNG wire#w7
   // the same network as SCL:
   #Dose_ChiliAwetan2.ISTART_AUT := #AlwaysON AND (#State."DoseHead1 ON" OR #State."DoseHead2 ON") AND #Dose.Dose_Tank_Available.%X1 AND (#Dose_ChiliAwetan2.SP_DOSEQTY > 0.0) AND NOT "AlarmFlowColletor".AlarmFlow_Blend.%X1 AND #Dose.Dose_Start.%X1;
   IF #AlwaysON AND ((NOT #State."DoseHead1 ON" AND NOT #State."DoseHead2 ON") OR NOT #Dose.Dose_Tank_Available.%X1) THEN
       #Dose.Dose_Start.%X1 := FALSE;
   END_IF;
   #Dose_ChiliAwetan2.IHOLD_AUT := #AlwaysON AND (#Dose.Dose_Pause.%X1 OR NOT #State."Dose EN" OR NOT #Dose.Dose_Prod_Ready.%X1 OR (NOT #State."DoseHead1 ON" AND NOT #State."DoseHead2 ON") OR "AlarmFlowColletor".AlarmFlow_Blend.%X1);
   #Dose_ChiliAwetan2.ISTOP_AUT := #AlwaysON AND (#Dose.Dose_Stop.%X1 OR ((NOT #State."Dose EN" OR NOT #Dose.Dose_Prod_Ready.%X1) AND #Dose_ChiliAwetan2.QHELD));
   #Dose_ChiliAwetan2.ICOMP_AUT := #AlwaysON AND (#Dose_ChiliAwetan2.QDoseComplete OR #Dose_ChiliAwetan2.QSTOPPED);
END_REGION

REGION Network 44: Dose ChiliAwetan2
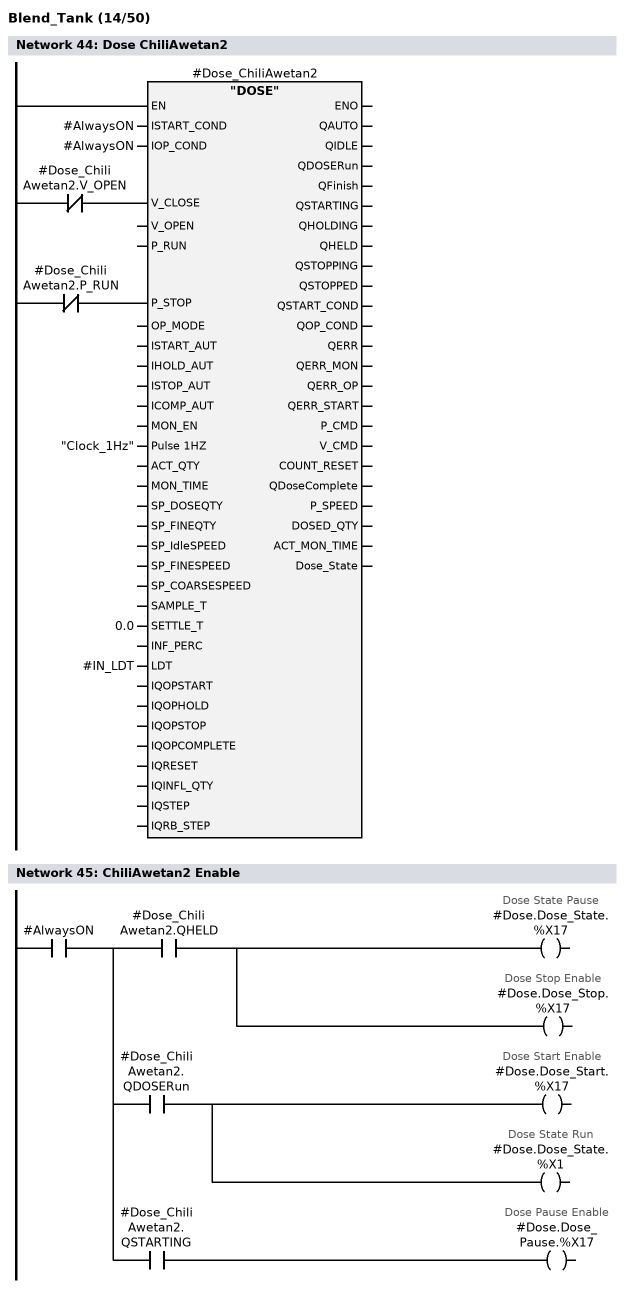
   RUNG wire#powerrail
      #Dose_ChiliAwetan2(V_CLOSE := wire#w1, P_STOP := wire#w2, ISTART_COND := #AlwaysON, IOP_COND := #AlwaysON, V_OPEN :=, P_RUN :=, OP_MODE :=, ISTART_AUT :=, IHOLD_AUT :=, ISTOP_AUT :=, ICOMP_AUT :=, MON_EN :=, "Pulse 1HZ" := "Clock_1Hz", ACT_QTY :=, MON_TIME :=, SP_DOSEQTY :=, SP_FINEQTY :=, SP_IdleSPEED :=, SP_FINESPEED :=, SP_COARSESPEED :=, SAMPLE_T :=, SETTLE_T := 0.0, INF_PERC :=, LDT := #IN_LDT, IQOPSTART :=, IQOPHOLD :=, IQOPSTOP :=, IQOPCOMPLETE :=, IQRESET :=, IQINFL_QTY :=, IQSTEP :=, IQRB_STEP :=, QAUTO =>, QIDLE =>, QDOSERun =>, QFinish =>, QSTARTING =>, QHOLDING =>, QHELD =>, QSTOPPING =>, QSTOPPED =>, QSTART_COND =>, QOP_COND =>, QERR =>, QERR_MON =>, QERR_OP =>, QERR_START =>, P_CMD =>, V_CMD =>, COUNT_RESET =>, QDoseComplete =>, P_SPEED =>, DOSED_QTY =>, ACT_MON_TIME =>, Dose_State =>)
   END_RUNG
   RUNG wire#powerrail
      I_Contact( #Dose_ChiliAwetan2.V_OPEN )
   END_RUNG wire#w1
   RUNG wire#powerrail
      I_Contact( #Dose_ChiliAwetan2.P_RUN )
   END_RUNG wire#w2
   // the same network as SCL:
   #Dose_ChiliAwetan2(ISTART_COND := #AlwaysON,   // "DOSE"
                      IOP_COND := #AlwaysON,
                      V_CLOSE := NOT #Dose_ChiliAwetan2.V_OPEN,
                      P_STOP := NOT #Dose_ChiliAwetan2.P_RUN,
                      "Pulse 1HZ" := "Clock_1Hz",
                      SETTLE_T := 0.0,
                      LDT := #IN_LDT);
END_REGION

REGION Network 45: ChiliAwetan2 Enable
   RUNG wire#powerrail
      Contact( #AlwaysON )
      wire#w1
      Contact( #Dose_ChiliAwetan2.QHELD )
      wire#w2
      Coil( #Dose.Dose_State.%X17 )   // Dose State Pause
   END_RUNG
   RUNG wire#w2
      Coil( #Dose.Dose_Stop.%X17 )   // Dose Stop Enable
   END_RUNG
   RUNG wire#w1
      Contact( #Dose_ChiliAwetan2.QDOSERun )
      wire#w3
      Coil( #Dose.Dose_Start.%X17 )   // Dose Start Enable
   END_RUNG
   RUNG wire#w3
      Coil( #Dose.Dose_State.%X1 )   // Dose State Run
   END_RUNG
   RUNG wire#w1
      Contact( #Dose_ChiliAwetan2.QSTARTING )
      Coil( #Dose.Dose_Pause.%X17 )   // Dose Pause Enable
   END_RUNG
   // the same network as SCL:
   #Dose.Dose_State.%X17 := #AlwaysON AND #Dose_ChiliAwetan2.QHELD;   // Dose State Pause
   #Dose.Dose_Stop.%X17 := #Dose.Dose_State.%X17;   // Dose Stop Enable
   #Dose.Dose_Start.%X17 := #AlwaysON AND #Dose_ChiliAwetan2.QDOSERun;   // Dose Start Enable
   #Dose.Dose_State.%X1 := #Dose.Dose_Start.%X17;   // Dose State Run
   #Dose.Dose_Pause.%X17 := #AlwaysON AND #Dose_ChiliAwetan2.QSTARTING;   // Dose Pause Enable
END_REGION

REGION Network 46: ChiliAwetan2 Header Req
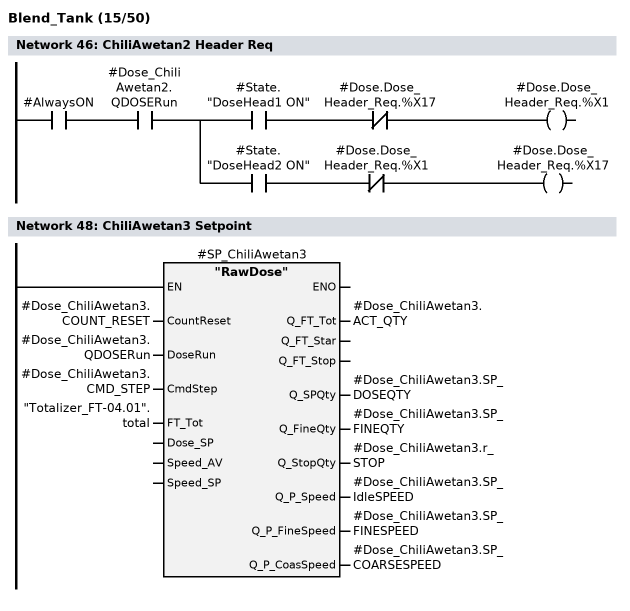
   RUNG wire#powerrail
      Contact( #AlwaysON )
      Contact( #Dose_ChiliAwetan2.QDOSERun )
      wire#w1
      Contact( #State."DoseHead1 ON" )
      I_Contact( #Dose.Dose_Header_Req.%X17 )
      Coil( #Dose.Dose_Header_Req.%X1 )
   END_RUNG
   RUNG wire#w1
      Contact( #State."DoseHead2 ON" )
      I_Contact( #Dose.Dose_Header_Req.%X1 )
      Coil( #Dose.Dose_Header_Req.%X17 )
   END_RUNG
   // the same network as SCL:
   #_w1 := #AlwaysON AND #Dose_ChiliAwetan2.QDOSERun;
   #Dose.Dose_Header_Req.%X1 := #_w1 AND #State."DoseHead1 ON" AND NOT #Dose.Dose_Header_Req.%X17;
   #Dose.Dose_Header_Req.%X17 := #_w1 AND #State."DoseHead2 ON" AND NOT #Dose.Dose_Header_Req.%X1;
END_REGION

REGION Network 48: ChiliAwetan3 Setpoint
   RUNG wire#powerrail
      #SP_ChiliAwetan3(CountReset := #Dose_ChiliAwetan3.COUNT_RESET, DoseRun := #Dose_ChiliAwetan3.QDOSERun, CmdStep := #Dose_ChiliAwetan3.CMD_STEP, FT_Tot := "Totalizer_FT-04.01".total, Dose_SP :=, Speed_AV :=, Speed_SP :=, Q_FT_Tot => #Dose_ChiliAwetan3.ACT_QTY, Q_FT_Star =>, Q_FT_Stop =>, Q_SPQty => #Dose_ChiliAwetan3.SP_DOSEQTY, Q_FineQty => #Dose_ChiliAwetan3.SP_FINEQTY, Q_StopQty => #Dose_ChiliAwetan3.r_STOP, Q_P_Speed => #Dose_ChiliAwetan3.SP_IdleSPEED, Q_P_FineSpeed => #Dose_ChiliAwetan3.SP_FINESPEED, Q_P_CoasSpeed => #Dose_ChiliAwetan3.SP_COARSESPEED)
   END_RUNG
   // the same network as SCL:
   #SP_ChiliAwetan3(CountReset := #Dose_ChiliAwetan3.COUNT_RESET,   // "RawDose"
                    DoseRun := #Dose_ChiliAwetan3.QDOSERun,
                    CmdStep := #Dose_ChiliAwetan3.CMD_STEP,
                    FT_Tot := "Totalizer_FT-04.01".total,
                    Q_FT_Tot => #Dose_ChiliAwetan3.ACT_QTY,
                    Q_SPQty => #Dose_ChiliAwetan3.SP_DOSEQTY,
                    Q_FineQty => #Dose_ChiliAwetan3.SP_FINEQTY,
                    Q_StopQty => #Dose_ChiliAwetan3.r_STOP,
                    Q_P_Speed => #Dose_ChiliAwetan3.SP_IdleSPEED,
                    Q_P_FineSpeed => #Dose_ChiliAwetan3.SP_FINESPEED,
                    Q_P_CoasSpeed => #Dose_ChiliAwetan3.SP_COARSESPEED);
END_REGION

REGION Network 49: Command Dose ChiliAwetan3
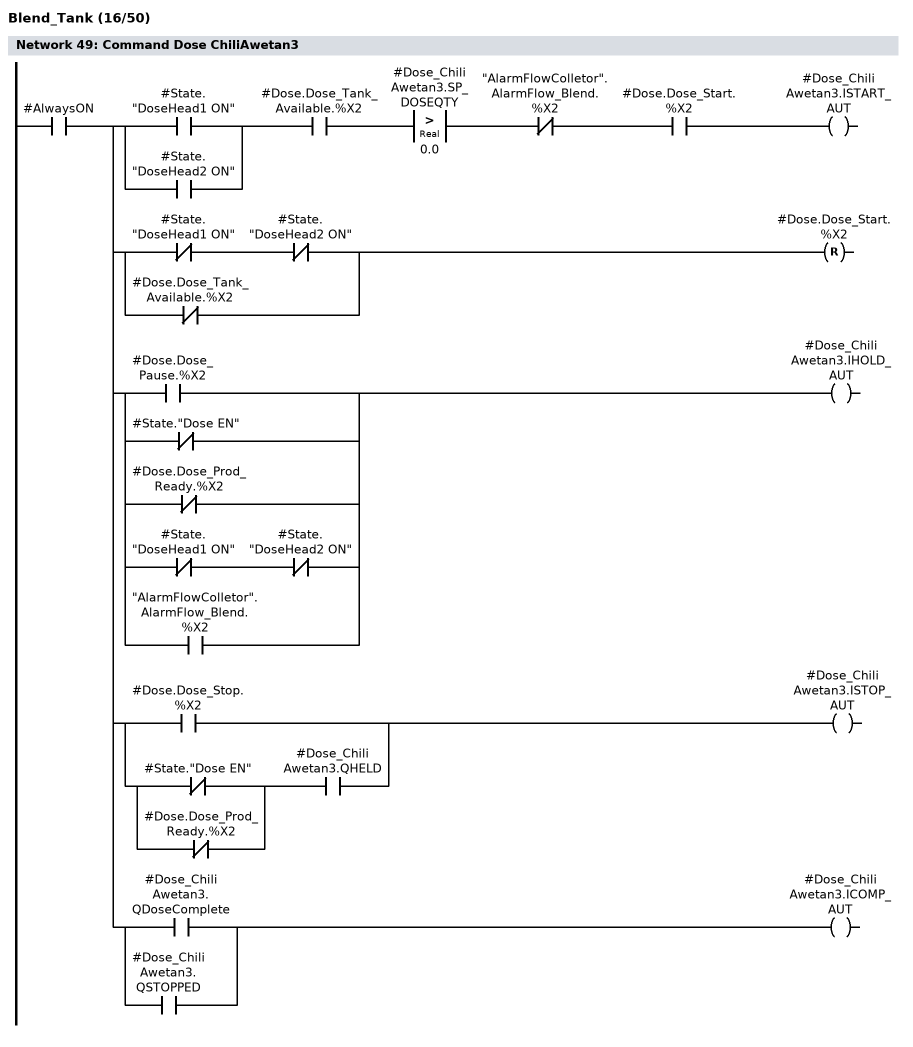
   RUNG wire#powerrail
      Contact( #AlwaysON )
      wire#w1
      Contact( #State."DoseHead1 ON" )
      wire#w2
      Contact( #Dose.Dose_Tank_Available.%X2 )
      { S7_Templates := "SrcType := Real" } GT_Contact(in1 := #Dose_ChiliAwetan3.SP_DOSEQTY, in2 := 0.0)
      I_Contact( "AlarmFlowColletor".AlarmFlow_Blend.%X2 )
      Contact( #Dose.Dose_Start.%X2 )
      Coil( #Dose_ChiliAwetan3.ISTART_AUT )
   END_RUNG
   RUNG wire#w1
      Contact( #State."DoseHead2 ON" )
   END_RUNG wire#w2
   RUNG wire#w1
      I_Contact( #State."DoseHead1 ON" )
      I_Contact( #State."DoseHead2 ON" )
      wire#w3
      R_Coil( #Dose.Dose_Start.%X2 )
   END_RUNG
   RUNG wire#w1
      I_Contact( #Dose.Dose_Tank_Available.%X2 )
   END_RUNG wire#w3
   RUNG wire#w1
      Contact( #Dose.Dose_Pause.%X2 )
      wire#w4
      Coil( #Dose_ChiliAwetan3.IHOLD_AUT )
   END_RUNG
   RUNG wire#w1
      I_Contact( #State."Dose EN" )
   END_RUNG wire#w4
   RUNG wire#w1
      I_Contact( #Dose.Dose_Prod_Ready.%X2 )
   END_RUNG wire#w4
   RUNG wire#w1
      I_Contact( #State."DoseHead1 ON" )
      I_Contact( #State."DoseHead2 ON" )
   END_RUNG wire#w4
   RUNG wire#w1
      Contact( "AlarmFlowColletor".AlarmFlow_Blend.%X2 )
   END_RUNG wire#w4
   RUNG wire#w1
      Contact( #Dose.Dose_Stop.%X2 )
      wire#w5
      Coil( #Dose_ChiliAwetan3.ISTOP_AUT )
   END_RUNG
   RUNG wire#w1
      I_Contact( #State."Dose EN" )
      wire#w6
      Contact( #Dose_ChiliAwetan3.QHELD )
   END_RUNG wire#w5
   RUNG wire#w1
      I_Contact( #Dose.Dose_Prod_Ready.%X2 )
   END_RUNG wire#w6
   RUNG wire#w1
      Contact( #Dose_ChiliAwetan3.QDoseComplete )
      wire#w7
      Coil( #Dose_ChiliAwetan3.ICOMP_AUT )
   END_RUNG
   RUNG wire#w1
      Contact( #Dose_ChiliAwetan3.QSTOPPED )
   END_RUNG wire#w7
   // the same network as SCL:
   #Dose_ChiliAwetan3.ISTART_AUT := #AlwaysON AND (#State."DoseHead1 ON" OR #State."DoseHead2 ON") AND #Dose.Dose_Tank_Available.%X2 AND (#Dose_ChiliAwetan3.SP_DOSEQTY > 0.0) AND NOT "AlarmFlowColletor".AlarmFlow_Blend.%X2 AND #Dose.Dose_Start.%X2;
   IF #AlwaysON AND ((NOT #State."DoseHead1 ON" AND NOT #State."DoseHead2 ON") OR NOT #Dose.Dose_Tank_Available.%X2) THEN
       #Dose.Dose_Start.%X2 := FALSE;
   END_IF;
   #Dose_ChiliAwetan3.IHOLD_AUT := #AlwaysON AND (#Dose.Dose_Pause.%X2 OR NOT #State."Dose EN" OR NOT #Dose.Dose_Prod_Ready.%X2 OR (NOT #State."DoseHead1 ON" AND NOT #State."DoseHead2 ON") OR "AlarmFlowColletor".AlarmFlow_Blend.%X2);
   #Dose_ChiliAwetan3.ISTOP_AUT := #AlwaysON AND (#Dose.Dose_Stop.%X2 OR ((NOT #State."Dose EN" OR NOT #Dose.Dose_Prod_Ready.%X2) AND #Dose_ChiliAwetan3.QHELD));
   #Dose_ChiliAwetan3.ICOMP_AUT := #AlwaysON AND (#Dose_ChiliAwetan3.QDoseComplete OR #Dose_ChiliAwetan3.QSTOPPED);
END_REGION

REGION Network 50: Dose ChiliAwetan3
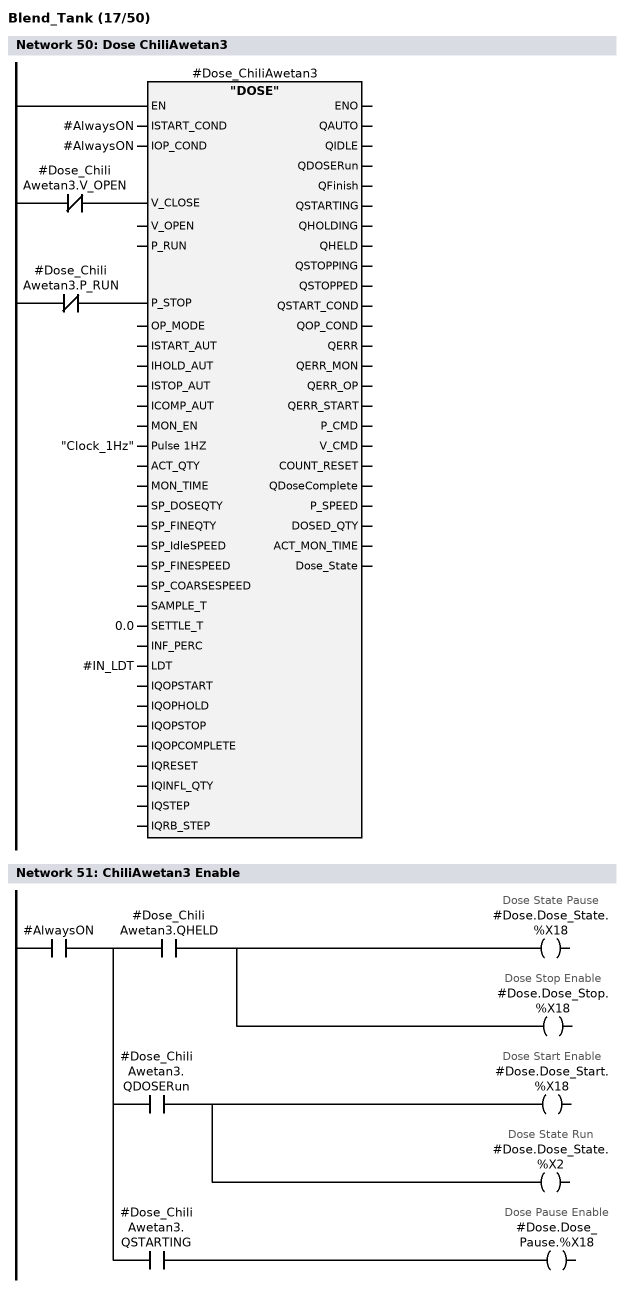
   RUNG wire#powerrail
      #Dose_ChiliAwetan3(V_CLOSE := wire#w1, P_STOP := wire#w2, ISTART_COND := #AlwaysON, IOP_COND := #AlwaysON, V_OPEN :=, P_RUN :=, OP_MODE :=, ISTART_AUT :=, IHOLD_AUT :=, ISTOP_AUT :=, ICOMP_AUT :=, MON_EN :=, "Pulse 1HZ" := "Clock_1Hz", ACT_QTY :=, MON_TIME :=, SP_DOSEQTY :=, SP_FINEQTY :=, SP_IdleSPEED :=, SP_FINESPEED :=, SP_COARSESPEED :=, SAMPLE_T :=, SETTLE_T := 0.0, INF_PERC :=, LDT := #IN_LDT, IQOPSTART :=, IQOPHOLD :=, IQOPSTOP :=, IQOPCOMPLETE :=, IQRESET :=, IQINFL_QTY :=, IQSTEP :=, IQRB_STEP :=, QAUTO =>, QIDLE =>, QDOSERun =>, QFinish =>, QSTARTING =>, QHOLDING =>, QHELD =>, QSTOPPING =>, QSTOPPED =>, QSTART_COND =>, QOP_COND =>, QERR =>, QERR_MON =>, QERR_OP =>, QERR_START =>, P_CMD =>, V_CMD =>, COUNT_RESET =>, QDoseComplete =>, P_SPEED =>, DOSED_QTY =>, ACT_MON_TIME =>, Dose_State =>)
   END_RUNG
   RUNG wire#powerrail
      I_Contact( #Dose_ChiliAwetan3.V_OPEN )
   END_RUNG wire#w1
   RUNG wire#powerrail
      I_Contact( #Dose_ChiliAwetan3.P_RUN )
   END_RUNG wire#w2
   // the same network as SCL:
   #Dose_ChiliAwetan3(ISTART_COND := #AlwaysON,   // "DOSE"
                      IOP_COND := #AlwaysON,
                      V_CLOSE := NOT #Dose_ChiliAwetan3.V_OPEN,
                      P_STOP := NOT #Dose_ChiliAwetan3.P_RUN,
                      "Pulse 1HZ" := "Clock_1Hz",
                      SETTLE_T := 0.0,
                      LDT := #IN_LDT);
END_REGION

REGION Network 51: ChiliAwetan3 Enable
   RUNG wire#powerrail
      Contact( #AlwaysON )
      wire#w1
      Contact( #Dose_ChiliAwetan3.QHELD )
      wire#w2
      Coil( #Dose.Dose_State.%X18 )   // Dose State Pause
   END_RUNG
   RUNG wire#w2
      Coil( #Dose.Dose_Stop.%X18 )   // Dose Stop Enable
   END_RUNG
   RUNG wire#w1
      Contact( #Dose_ChiliAwetan3.QDOSERun )
      wire#w3
      Coil( #Dose.Dose_Start.%X18 )   // Dose Start Enable
   END_RUNG
   RUNG wire#w3
      Coil( #Dose.Dose_State.%X2 )   // Dose State Run
   END_RUNG
   RUNG wire#w1
      Contact( #Dose_ChiliAwetan3.QSTARTING )
      Coil( #Dose.Dose_Pause.%X18 )   // Dose Pause Enable
   END_RUNG
   // the same network as SCL:
   #Dose.Dose_State.%X18 := #AlwaysON AND #Dose_ChiliAwetan3.QHELD;   // Dose State Pause
   #Dose.Dose_Stop.%X18 := #Dose.Dose_State.%X18;   // Dose Stop Enable
   #Dose.Dose_Start.%X18 := #AlwaysON AND #Dose_ChiliAwetan3.QDOSERun;   // Dose Start Enable
   #Dose.Dose_State.%X2 := #Dose.Dose_Start.%X18;   // Dose State Run
   #Dose.Dose_Pause.%X18 := #AlwaysON AND #Dose_ChiliAwetan3.QSTARTING;   // Dose Pause Enable
END_REGION

REGION Network 52: ChiliAwetan3 Header Req
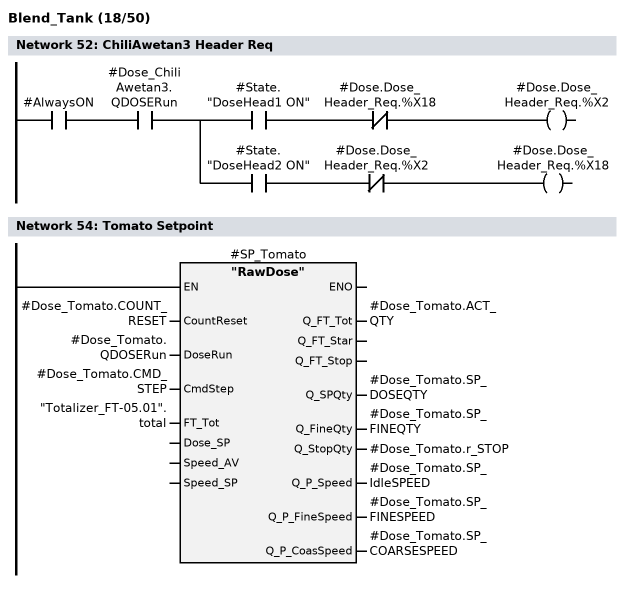
   RUNG wire#powerrail
      Contact( #AlwaysON )
      Contact( #Dose_ChiliAwetan3.QDOSERun )
      wire#w1
      Contact( #State."DoseHead1 ON" )
      I_Contact( #Dose.Dose_Header_Req.%X18 )
      Coil( #Dose.Dose_Header_Req.%X2 )
   END_RUNG
   RUNG wire#w1
      Contact( #State."DoseHead2 ON" )
      I_Contact( #Dose.Dose_Header_Req.%X2 )
      Coil( #Dose.Dose_Header_Req.%X18 )
   END_RUNG
   // the same network as SCL:
   #_w1 := #AlwaysON AND #Dose_ChiliAwetan3.QDOSERun;
   #Dose.Dose_Header_Req.%X2 := #_w1 AND #State."DoseHead1 ON" AND NOT #Dose.Dose_Header_Req.%X18;
   #Dose.Dose_Header_Req.%X18 := #_w1 AND #State."DoseHead2 ON" AND NOT #Dose.Dose_Header_Req.%X2;
END_REGION

REGION Network 54: Tomato Setpoint
   RUNG wire#powerrail
      #SP_Tomato(CountReset := #Dose_Tomato.COUNT_RESET, DoseRun := #Dose_Tomato.QDOSERun, CmdStep := #Dose_Tomato.CMD_STEP, FT_Tot := "Totalizer_FT-05.01".total, Dose_SP :=, Speed_AV :=, Speed_SP :=, Q_FT_Tot => #Dose_Tomato.ACT_QTY, Q_FT_Star =>, Q_FT_Stop =>, Q_SPQty => #Dose_Tomato.SP_DOSEQTY, Q_FineQty => #Dose_Tomato.SP_FINEQTY, Q_StopQty => #Dose_Tomato.r_STOP, Q_P_Speed => #Dose_Tomato.SP_IdleSPEED, Q_P_FineSpeed => #Dose_Tomato.SP_FINESPEED, Q_P_CoasSpeed => #Dose_Tomato.SP_COARSESPEED)
   END_RUNG
   // the same network as SCL:
   #SP_Tomato(CountReset := #Dose_Tomato.COUNT_RESET,   // "RawDose"
              DoseRun := #Dose_Tomato.QDOSERun,
              CmdStep := #Dose_Tomato.CMD_STEP,
              FT_Tot := "Totalizer_FT-05.01".total,
              Q_FT_Tot => #Dose_Tomato.ACT_QTY,
              Q_SPQty => #Dose_Tomato.SP_DOSEQTY,
              Q_FineQty => #Dose_Tomato.SP_FINEQTY,
              Q_StopQty => #Dose_Tomato.r_STOP,
              Q_P_Speed => #Dose_Tomato.SP_IdleSPEED,
              Q_P_FineSpeed => #Dose_Tomato.SP_FINESPEED,
              Q_P_CoasSpeed => #Dose_Tomato.SP_COARSESPEED);
END_REGION

REGION Network 55: Command Dose Tomato
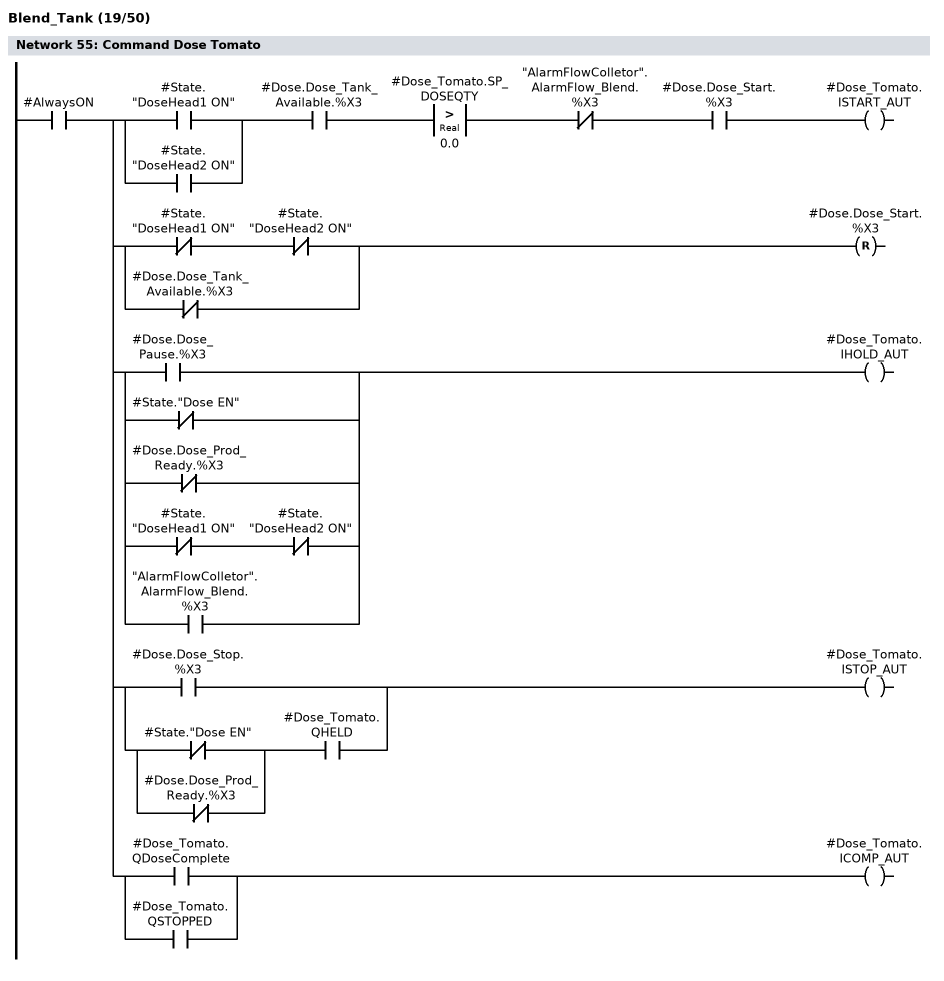
   RUNG wire#powerrail
      Contact( #AlwaysON )
      wire#w1
      Contact( #State."DoseHead1 ON" )
      wire#w2
      Contact( #Dose.Dose_Tank_Available.%X3 )
      { S7_Templates := "SrcType := Real" } GT_Contact(in1 := #Dose_Tomato.SP_DOSEQTY, in2 := 0.0)
      I_Contact( "AlarmFlowColletor".AlarmFlow_Blend.%X3 )
      Contact( #Dose.Dose_Start.%X3 )
      Coil( #Dose_Tomato.ISTART_AUT )
   END_RUNG
   RUNG wire#w1
      Contact( #State."DoseHead2 ON" )
   END_RUNG wire#w2
   RUNG wire#w1
      I_Contact( #State."DoseHead1 ON" )
      I_Contact( #State."DoseHead2 ON" )
      wire#w3
      R_Coil( #Dose.Dose_Start.%X3 )
   END_RUNG
   RUNG wire#w1
      I_Contact( #Dose.Dose_Tank_Available.%X3 )
   END_RUNG wire#w3
   RUNG wire#w1
      Contact( #Dose.Dose_Pause.%X3 )
      wire#w4
      Coil( #Dose_Tomato.IHOLD_AUT )
   END_RUNG
   RUNG wire#w1
      I_Contact( #State."Dose EN" )
   END_RUNG wire#w4
   RUNG wire#w1
      I_Contact( #Dose.Dose_Prod_Ready.%X3 )
   END_RUNG wire#w4
   RUNG wire#w1
      I_Contact( #State."DoseHead1 ON" )
      I_Contact( #State."DoseHead2 ON" )
   END_RUNG wire#w4
   RUNG wire#w1
      Contact( "AlarmFlowColletor".AlarmFlow_Blend.%X3 )
   END_RUNG wire#w4
   RUNG wire#w1
      Contact( #Dose.Dose_Stop.%X3 )
      wire#w5
      Coil( #Dose_Tomato.ISTOP_AUT )
   END_RUNG
   RUNG wire#w1
      I_Contact( #State."Dose EN" )
      wire#w6
      Contact( #Dose_Tomato.QHELD )
   END_RUNG wire#w5
   RUNG wire#w1
      I_Contact( #Dose.Dose_Prod_Ready.%X3 )
   END_RUNG wire#w6
   RUNG wire#w1
      Contact( #Dose_Tomato.QDoseComplete )
      wire#w7
      Coil( #Dose_Tomato.ICOMP_AUT )
   END_RUNG
   RUNG wire#w1
      Contact( #Dose_Tomato.QSTOPPED )
   END_RUNG wire#w7
   // the same network as SCL:
   #Dose_Tomato.ISTART_AUT := #AlwaysON AND (#State."DoseHead1 ON" OR #State."DoseHead2 ON") AND #Dose.Dose_Tank_Available.%X3 AND (#Dose_Tomato.SP_DOSEQTY > 0.0) AND NOT "AlarmFlowColletor".AlarmFlow_Blend.%X3 AND #Dose.Dose_Start.%X3;
   IF #AlwaysON AND ((NOT #State."DoseHead1 ON" AND NOT #State."DoseHead2 ON") OR NOT #Dose.Dose_Tank_Available.%X3) THEN
       #Dose.Dose_Start.%X3 := FALSE;
   END_IF;
   #Dose_Tomato.IHOLD_AUT := #AlwaysON AND (#Dose.Dose_Pause.%X3 OR NOT #State."Dose EN" OR NOT #Dose.Dose_Prod_Ready.%X3 OR (NOT #State."DoseHead1 ON" AND NOT #State."DoseHead2 ON") OR "AlarmFlowColletor".AlarmFlow_Blend.%X3);
   #Dose_Tomato.ISTOP_AUT := #AlwaysON AND (#Dose.Dose_Stop.%X3 OR ((NOT #State."Dose EN" OR NOT #Dose.Dose_Prod_Ready.%X3) AND #Dose_Tomato.QHELD));
   #Dose_Tomato.ICOMP_AUT := #AlwaysON AND (#Dose_Tomato.QDoseComplete OR #Dose_Tomato.QSTOPPED);
END_REGION

REGION Network 56: Dose Tomato
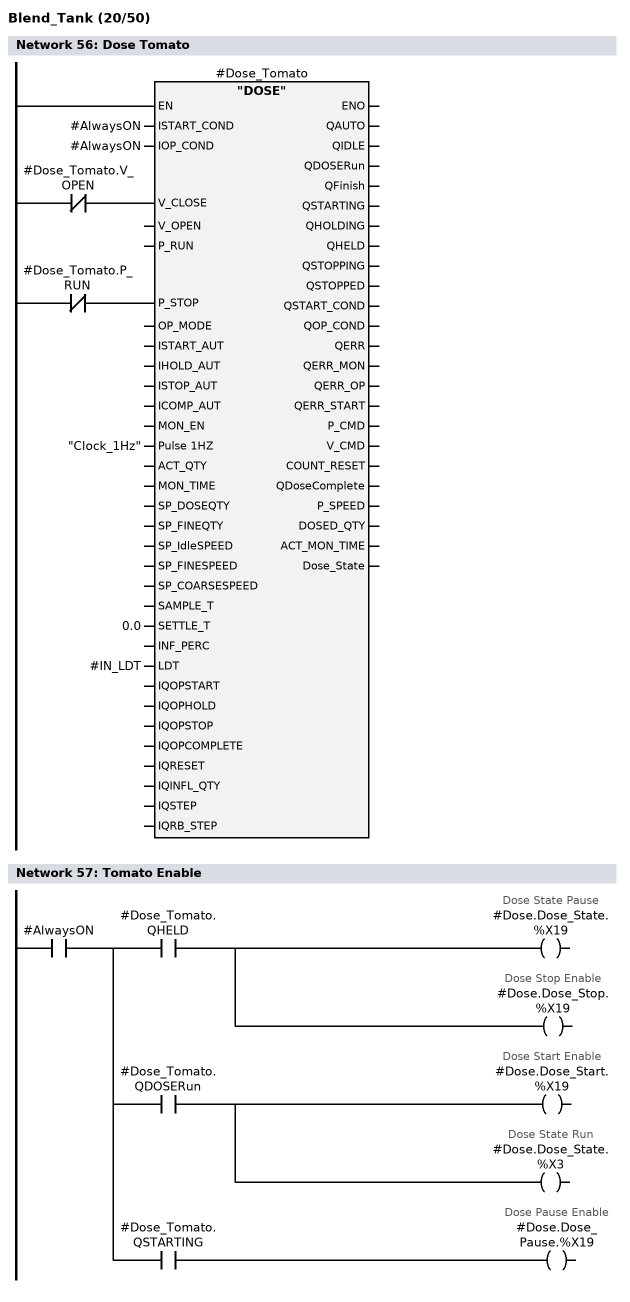
   RUNG wire#powerrail
      #Dose_Tomato(V_CLOSE := wire#w1, P_STOP := wire#w2, ISTART_COND := #AlwaysON, IOP_COND := #AlwaysON, V_OPEN :=, P_RUN :=, OP_MODE :=, ISTART_AUT :=, IHOLD_AUT :=, ISTOP_AUT :=, ICOMP_AUT :=, MON_EN :=, "Pulse 1HZ" := "Clock_1Hz", ACT_QTY :=, MON_TIME :=, SP_DOSEQTY :=, SP_FINEQTY :=, SP_IdleSPEED :=, SP_FINESPEED :=, SP_COARSESPEED :=, SAMPLE_T :=, SETTLE_T := 0.0, INF_PERC :=, LDT := #IN_LDT, IQOPSTART :=, IQOPHOLD :=, IQOPSTOP :=, IQOPCOMPLETE :=, IQRESET :=, IQINFL_QTY :=, IQSTEP :=, IQRB_STEP :=, QAUTO =>, QIDLE =>, QDOSERun =>, QFinish =>, QSTARTING =>, QHOLDING =>, QHELD =>, QSTOPPING =>, QSTOPPED =>, QSTART_COND =>, QOP_COND =>, QERR =>, QERR_MON =>, QERR_OP =>, QERR_START =>, P_CMD =>, V_CMD =>, COUNT_RESET =>, QDoseComplete =>, P_SPEED =>, DOSED_QTY =>, ACT_MON_TIME =>, Dose_State =>)
   END_RUNG
   RUNG wire#powerrail
      I_Contact( #Dose_Tomato.V_OPEN )
   END_RUNG wire#w1
   RUNG wire#powerrail
      I_Contact( #Dose_Tomato.P_RUN )
   END_RUNG wire#w2
   // the same network as SCL:
   #Dose_Tomato(ISTART_COND := #AlwaysON,   // "DOSE"
                IOP_COND := #AlwaysON,
                V_CLOSE := NOT #Dose_Tomato.V_OPEN,
                P_STOP := NOT #Dose_Tomato.P_RUN,
                "Pulse 1HZ" := "Clock_1Hz",
                SETTLE_T := 0.0,
                LDT := #IN_LDT);
END_REGION

REGION Network 57: Tomato Enable
   RUNG wire#powerrail
      Contact( #AlwaysON )
      wire#w1
      Contact( #Dose_Tomato.QHELD )
      wire#w2
      Coil( #Dose.Dose_State.%X19 )   // Dose State Pause
   END_RUNG
   RUNG wire#w2
      Coil( #Dose.Dose_Stop.%X19 )   // Dose Stop Enable
   END_RUNG
   RUNG wire#w1
      Contact( #Dose_Tomato.QDOSERun )
      wire#w3
      Coil( #Dose.Dose_Start.%X19 )   // Dose Start Enable
   END_RUNG
   RUNG wire#w3
      Coil( #Dose.Dose_State.%X3 )   // Dose State Run
   END_RUNG
   RUNG wire#w1
      Contact( #Dose_Tomato.QSTARTING )
      Coil( #Dose.Dose_Pause.%X19 )   // Dose Pause Enable
   END_RUNG
   // the same network as SCL:
   #Dose.Dose_State.%X19 := #AlwaysON AND #Dose_Tomato.QHELD;   // Dose State Pause
   #Dose.Dose_Stop.%X19 := #Dose.Dose_State.%X19;   // Dose Stop Enable
   #Dose.Dose_Start.%X19 := #AlwaysON AND #Dose_Tomato.QDOSERun;   // Dose Start Enable
   #Dose.Dose_State.%X3 := #Dose.Dose_Start.%X19;   // Dose State Run
   #Dose.Dose_Pause.%X19 := #AlwaysON AND #Dose_Tomato.QSTARTING;   // Dose Pause Enable
END_REGION

REGION Network 58: Tomato Header Req
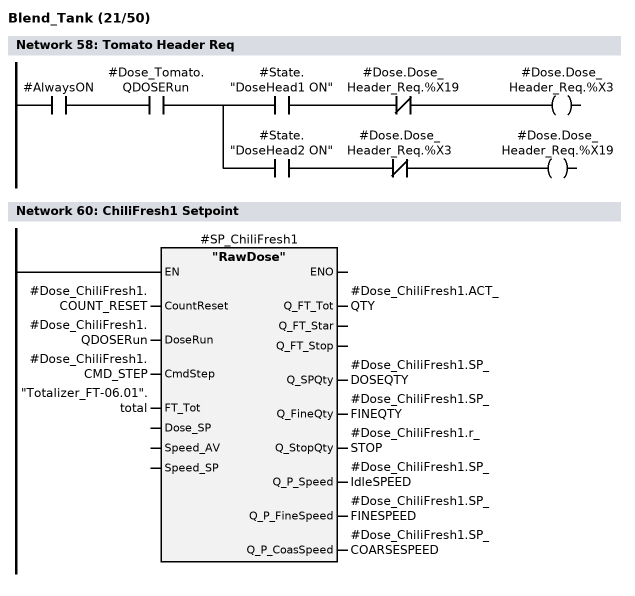
   RUNG wire#powerrail
      Contact( #AlwaysON )
      Contact( #Dose_Tomato.QDOSERun )
      wire#w1
      Contact( #State."DoseHead1 ON" )
      I_Contact( #Dose.Dose_Header_Req.%X19 )
      Coil( #Dose.Dose_Header_Req.%X3 )
   END_RUNG
   RUNG wire#w1
      Contact( #State."DoseHead2 ON" )
      I_Contact( #Dose.Dose_Header_Req.%X3 )
      Coil( #Dose.Dose_Header_Req.%X19 )
   END_RUNG
   // the same network as SCL:
   #_w1 := #AlwaysON AND #Dose_Tomato.QDOSERun;
   #Dose.Dose_Header_Req.%X3 := #_w1 AND #State."DoseHead1 ON" AND NOT #Dose.Dose_Header_Req.%X19;
   #Dose.Dose_Header_Req.%X19 := #_w1 AND #State."DoseHead2 ON" AND NOT #Dose.Dose_Header_Req.%X3;
END_REGION

REGION Network 60: ChiliFresh1 Setpoint
   RUNG wire#powerrail
      #SP_ChiliFresh1(CountReset := #Dose_ChiliFresh1.COUNT_RESET, DoseRun := #Dose_ChiliFresh1.QDOSERun, CmdStep := #Dose_ChiliFresh1.CMD_STEP, FT_Tot := "Totalizer_FT-06.01".total, Dose_SP :=, Speed_AV :=, Speed_SP :=, Q_FT_Tot => #Dose_ChiliFresh1.ACT_QTY, Q_FT_Star =>, Q_FT_Stop =>, Q_SPQty => #Dose_ChiliFresh1.SP_DOSEQTY, Q_FineQty => #Dose_ChiliFresh1.SP_FINEQTY, Q_StopQty => #Dose_ChiliFresh1.r_STOP, Q_P_Speed => #Dose_ChiliFresh1.SP_IdleSPEED, Q_P_FineSpeed => #Dose_ChiliFresh1.SP_FINESPEED, Q_P_CoasSpeed => #Dose_ChiliFresh1.SP_COARSESPEED)
   END_RUNG
   // the same network as SCL:
   #SP_ChiliFresh1(CountReset := #Dose_ChiliFresh1.COUNT_RESET,   // "RawDose"
                   DoseRun := #Dose_ChiliFresh1.QDOSERun,
                   CmdStep := #Dose_ChiliFresh1.CMD_STEP,
                   FT_Tot := "Totalizer_FT-06.01".total,
                   Q_FT_Tot => #Dose_ChiliFresh1.ACT_QTY,
                   Q_SPQty => #Dose_ChiliFresh1.SP_DOSEQTY,
                   Q_FineQty => #Dose_ChiliFresh1.SP_FINEQTY,
                   Q_StopQty => #Dose_ChiliFresh1.r_STOP,
                   Q_P_Speed => #Dose_ChiliFresh1.SP_IdleSPEED,
                   Q_P_FineSpeed => #Dose_ChiliFresh1.SP_FINESPEED,
                   Q_P_CoasSpeed => #Dose_ChiliFresh1.SP_COARSESPEED);
END_REGION

REGION Network 61: Command Dose ChiliFresh1
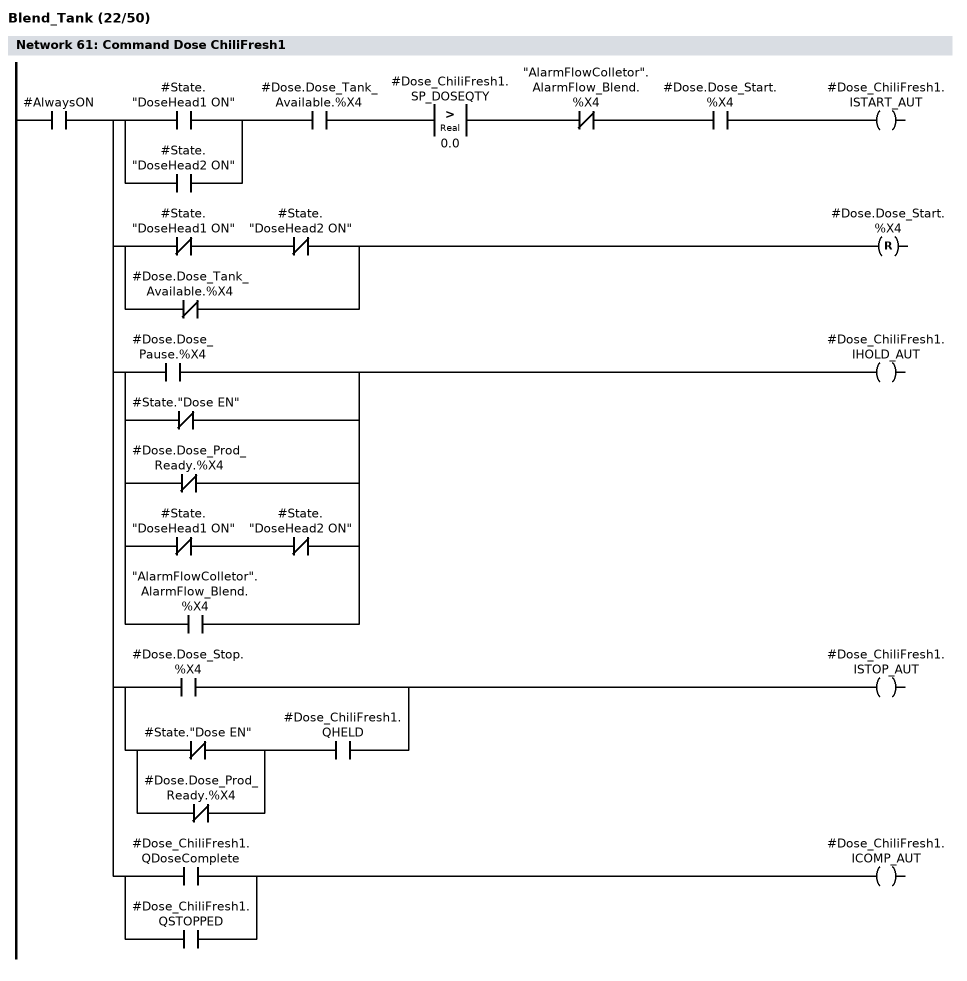
   RUNG wire#powerrail
      Contact( #AlwaysON )
      wire#w1
      Contact( #State."DoseHead1 ON" )
      wire#w2
      Contact( #Dose.Dose_Tank_Available.%X4 )
      { S7_Templates := "SrcType := Real" } GT_Contact(in1 := #Dose_ChiliFresh1.SP_DOSEQTY, in2 := 0.0)
      I_Contact( "AlarmFlowColletor".AlarmFlow_Blend.%X4 )
      Contact( #Dose.Dose_Start.%X4 )
      Coil( #Dose_ChiliFresh1.ISTART_AUT )
   END_RUNG
   RUNG wire#w1
      Contact( #State."DoseHead2 ON" )
   END_RUNG wire#w2
   RUNG wire#w1
      I_Contact( #State."DoseHead1 ON" )
      I_Contact( #State."DoseHead2 ON" )
      wire#w3
      R_Coil( #Dose.Dose_Start.%X4 )
   END_RUNG
   RUNG wire#w1
      I_Contact( #Dose.Dose_Tank_Available.%X4 )
   END_RUNG wire#w3
   RUNG wire#w1
      Contact( #Dose.Dose_Pause.%X4 )
      wire#w4
      Coil( #Dose_ChiliFresh1.IHOLD_AUT )
   END_RUNG
   RUNG wire#w1
      I_Contact( #State."Dose EN" )
   END_RUNG wire#w4
   RUNG wire#w1
      I_Contact( #Dose.Dose_Prod_Ready.%X4 )
   END_RUNG wire#w4
   RUNG wire#w1
      I_Contact( #State."DoseHead1 ON" )
      I_Contact( #State."DoseHead2 ON" )
   END_RUNG wire#w4
   RUNG wire#w1
      Contact( "AlarmFlowColletor".AlarmFlow_Blend.%X4 )
   END_RUNG wire#w4
   RUNG wire#w1
      Contact( #Dose.Dose_Stop.%X4 )
      wire#w5
      Coil( #Dose_ChiliFresh1.ISTOP_AUT )
   END_RUNG
   RUNG wire#w1
      I_Contact( #State."Dose EN" )
      wire#w6
      Contact( #Dose_ChiliFresh1.QHELD )
   END_RUNG wire#w5
   RUNG wire#w1
      I_Contact( #Dose.Dose_Prod_Ready.%X4 )
   END_RUNG wire#w6
   RUNG wire#w1
      Contact( #Dose_ChiliFresh1.QDoseComplete )
      wire#w7
      Coil( #Dose_ChiliFresh1.ICOMP_AUT )
   END_RUNG
   RUNG wire#w1
      Contact( #Dose_ChiliFresh1.QSTOPPED )
   END_RUNG wire#w7
   // the same network as SCL:
   #Dose_ChiliFresh1.ISTART_AUT := #AlwaysON AND (#State."DoseHead1 ON" OR #State."DoseHead2 ON") AND #Dose.Dose_Tank_Available.%X4 AND (#Dose_ChiliFresh1.SP_DOSEQTY > 0.0) AND NOT "AlarmFlowColletor".AlarmFlow_Blend.%X4 AND #Dose.Dose_Start.%X4;
   IF #AlwaysON AND ((NOT #State."DoseHead1 ON" AND NOT #State."DoseHead2 ON") OR NOT #Dose.Dose_Tank_Available.%X4) THEN
       #Dose.Dose_Start.%X4 := FALSE;
   END_IF;
   #Dose_ChiliFresh1.IHOLD_AUT := #AlwaysON AND (#Dose.Dose_Pause.%X4 OR NOT #State."Dose EN" OR NOT #Dose.Dose_Prod_Ready.%X4 OR (NOT #State."DoseHead1 ON" AND NOT #State."DoseHead2 ON") OR "AlarmFlowColletor".AlarmFlow_Blend.%X4);
   #Dose_ChiliFresh1.ISTOP_AUT := #AlwaysON AND (#Dose.Dose_Stop.%X4 OR ((NOT #State."Dose EN" OR NOT #Dose.Dose_Prod_Ready.%X4) AND #Dose_ChiliFresh1.QHELD));
   #Dose_ChiliFresh1.ICOMP_AUT := #AlwaysON AND (#Dose_ChiliFresh1.QDoseComplete OR #Dose_ChiliFresh1.QSTOPPED);
END_REGION

REGION Network 62: Dose ChiliFresh1
